// TwinCAT 3 PLC project PLC
// ProgramVersion: 3.1.4026.26
// libraries:
//   Tc2_Standard, * (Beckhoff Automation GmbH)
//   Tc2_System, * (Beckhoff Automation GmbH)
//   Tc2_Utilities, * (Beckhoff Automation GmbH)
//   Tc3_Database, * (Beckhoff Automation GmbH)
//   Tc3_EventLogger, * (Beckhoff Automation GmbH)
//   Tc3_JsonXml, * (Beckhoff Automation GmbH)
//   Tc3_IotBase, * (Beckhoff Automation GmbH)
//   TcUnit, * (www.tcunit.org)
// project tree:
//   / PlcTask.TcTTO, TestTask.TcTTO
//   POUs/ MAIN.TcPOU
//   POUs/fb/ FB_DfiRowBuffer.TcPOU, FB_DfiSampler.TcPOU, F_DfiNowString.TcPOU, FB_DfiCfgParse.TcPOU, FB_DfiConfigLoader.TcPOU, F_DfiSanitizeText.TcPOU, F_DfiStripSqlUnsafe.TcPOU, FB_DfiPayloadParser.TcPOU, FB_DfiSqlBuilder.TcPOU, FB_DfiDbWriter.TcPOU, FB_DfiMqttSubscriber.TcPOU
//   POUs/test/ PRG_DfiTests.TcPOU, FB_DfiRowBuffer_Tests.TcPOU, FB_DfiSampler_Tests.TcPOU, FB_DfiCfgParse_Tests.TcPOU, FB_DfiPayloadParser_Tests.TcPOU, FB_DfiSqlBuilder_Tests.TcPOU, F_DfiNowString_Tests.TcPOU, FB_DfiDbWriter_Fake.TcPOU, FB_DfiDbWriter_Tests.TcPOU
//   DUTs/ E_DfiRowKind.TcDUT, E_DfiWriterState.TcDUT, ST_EstoqueSnapshot.TcDUT, ST_EventoDfi.TcDUT, ST_DfiRow.TcDUT, ST_DfiConfig.TcDUT, ST_DfiDiag.TcDUT
//   GVLs/ GVL_Dfi.TcGVL
// real-time tasks:
//   TASK PlcTask: cycle T#100000us, priority 20, ADS port 350
//   TASK TestTask: cycle T#100000us, priority 21, ADS port 351

CONFIGURATION PLC
    RESOURCE PLC ON TwinCAT3
        TASK PlcTask(INTERVAL := T#10ms, PRIORITY := 1);
        TASK TestTask(INTERVAL := T#10ms, PRIORITY := 2);
        PROGRAM MAIN WITH PlcTask : MAIN;
        PROGRAM PRG_DfiTests WITH TestTask : PRG_DfiTests;
    END_RESOURCE
END_CONFIGURATION

// ---- DUTs/E_DfiRowKind.TcDUT
TYPE E_DfiRowKind :
(
	ESTOQUE_MUDANCA := 0,
	ESTOQUE_PERIODICO := 1,
	EVENTO := 2
) DINT;
END_TYPE

// ---- DUTs/E_DfiWriterState.TcDUT
TYPE E_DfiWriterState :
(
	IDLE := 0,
	CONNECT := 10,
	BUILD := 20,
	EXECUTE := 30,
	COMMIT := 40,
	ERROR := 90,
	DB_LOST := 99
) DINT;
END_TYPE

// ---- DUTs/ST_EstoqueSnapshot.TcDUT
TYPE ST_EstoqueSnapshot :
STRUCT
	nA : INT;
	nB : INT;
	nC : INT;
END_STRUCT
END_TYPE

// ---- DUTs/ST_EventoDfi.TcDUT
TYPE ST_EventoDfi :
STRUCT
	sEvento     : STRING(23);   // coluna eventos_hist.evento VARCHAR(24)
	sPeca       : STRING(1);    // 'A'|'B'|'C' ou '' (=> NULL)
	sDetalhe    : STRING(63);   // coluna detalhe VARCHAR(64)
	sPayloadRaw : STRING(254);  // coluna payload_raw VARCHAR(255)
END_STRUCT
END_TYPE

// ---- DUTs/ST_DfiRow.TcDUT
TYPE ST_DfiRow :
STRUCT
	eKind     : E_DfiRowKind;
	sTsPlc    : STRING(23);   // 'YYYY-MM-DD HH:MM:SS.mmm', carimbado no Push
	stEstoque : ST_EstoqueSnapshot;
	stEvento  : ST_EventoDfi;
END_STRUCT
END_TYPE

// ---- DUTs/ST_DfiConfig.TcDUT
TYPE ST_DfiConfig :
STRUCT
	sMqttHost     : STRING(120);
	nMqttPort     : UINT  := 1883;
	bUseTls       : BOOL  := FALSE;
	sCaCertPath   : STRING(255) := '/etc/ssl/certs/ca-certificates.crt';
	sMqttUser     : STRING(60);
	sMqttPass     : STRING(60);
	sTopicEstoque : STRING(120) := 'dataflow/estoque';
	sTopicEventos : STRING(120) := 'dataflow/eventos';
	nDbId         : UDINT := 1;
	tSamplePeriod : TIME  := T#60S;
	nBufferSize   : UDINT := 128;   // teto = FB_DfiRowBuffer.MAX_ROWS
	nEstoqueMax   : INT   := 999;
	bValid        : BOOL  := FALSE;   // TRUE após FB_DfiConfigLoader parsear o arquivo com sucesso
END_STRUCT
END_TYPE

// ---- DUTs/ST_DfiDiag.TcDUT
TYPE ST_DfiDiag :
STRUCT
	bConfigOk         : BOOL;
	bMqttConnected    : BOOL;
	bDbConnected      : BOOL;
	nReconnectCount   : UDINT;
	nBufferCount      : UDINT;
	nBufferHighWater  : UDINT;
	nBufferDropped    : ULINT;
	nRowsWritten      : ULINT;
	nDbErrors         : ULINT;
	nParseErrors      : ULINT;
	sUltimoParseError : STRING(120);
	sUltimoDbError    : STRING(255);
	eWriterState      : E_DfiWriterState;
END_STRUCT
END_TYPE

// ---- GVLs/GVL_Dfi.TcGVL
{attribute 'qualified_only'}
VAR_GLOBAL
	gCfg  : ST_DfiConfig;
	gDiag : ST_DfiDiag;
	// relogio de parede local (fonte do ts_plc; MAIN chama fbNow(bEnable := TRUE) todo ciclo)
	fbNow : Tc2_Utilities.FB_LocalSystemTime;
	// pipeline
	fbLoader  : FB_DfiConfigLoader;
	fbSub     : FB_DfiMqttSubscriber;
	fbParser  : FB_DfiPayloadParser;
	fbBuffer  : FB_DfiRowBuffer;
	fbSampler : FB_DfiSampler;
	fbWriter  : FB_DfiDbWriter;
END_VAR

// ---- POUs/MAIN.TcPOU
PROGRAM MAIN
VAR
	bBoot           : BOOL := TRUE;
	stUltimoEstoque : ST_EstoqueSnapshot;
	bEstoqueValido  : BOOL;
	bDiff           : BOOL;
	row             : ST_DfiRow;
END_VAR

// ---------------------------------------------------------------
// Orquestracao do historian DFI (Task 14). Pipeline por ciclo:
//   Config -> MQTT -> Parser -> Buffer -> Sampler -> DbWriter -> Diagnostico
// ---------------------------------------------------------------

// Relogio de parede local: ticado todo ciclo (independe da config) para que
// F_DfiNowString() tenha um TIMESTRUCT valido. Leva alguns ciclos ate bValid.
GVL_Dfi.fbNow(bEnable := TRUE);

// 0. Config (uma vez no arranque; retenta se falhar)
IF bBoot THEN
	GVL_Dfi.fbLoader(bExecute := TRUE, sPath := '/etc/dfi/historian.conf');
	IF GVL_Dfi.fbLoader.bDone THEN
		bBoot := FALSE;
		IF NOT GVL_Dfi.fbLoader.bError AND GVL_Dfi.fbLoader.stCfg.bValid THEN
			GVL_Dfi.gCfg := GVL_Dfi.fbLoader.stCfg;
		END_IF
	END_IF
END_IF
GVL_Dfi.gDiag.bConfigOk := GVL_Dfi.gCfg.bValid;
IF NOT GVL_Dfi.gCfg.bValid THEN
	RETURN;   // sem config valida, nao conecta em nada
END_IF

GVL_Dfi.fbBuffer(nCapacity := GVL_Dfi.gCfg.nBufferSize);

// 1. MQTT
GVL_Dfi.fbSub(stConfig := GVL_Dfi.gCfg, bEnable := TRUE);

// 2. Parse + roteamento
IF GVL_Dfi.fbSub.bNewMessage THEN
	GVL_Dfi.fbParser(bExecute := TRUE,
	                 sTopic   := GVL_Dfi.fbSub.sTopic,
	                 sPayload := GVL_Dfi.fbSub.sPayload,
	                 stConfig := GVL_Dfi.gCfg);
	IF GVL_Dfi.fbParser.bOk THEN
		// Limpa a linha reutilizada antes de montar (row e VAR persistente do MAIN).
		row.sTsPlc              := '';
		row.stEstoque.nA        := 0;
		row.stEstoque.nB        := 0;
		row.stEstoque.nC        := 0;
		row.stEvento.sEvento    := '';
		row.stEvento.sPeca      := '';
		row.stEvento.sDetalhe   := '';
		row.stEvento.sPayloadRaw := '';
		CASE GVL_Dfi.fbParser.eKind OF
			E_DfiRowKind.ESTOQUE_MUDANCA:
				stUltimoEstoque := GVL_Dfi.fbParser.stEstoque;
				bEstoqueValido  := TRUE;
				bDiff := (NOT GVL_Dfi.fbWriter.bUltimoGravadoValido)
				      OR (GVL_Dfi.fbParser.stEstoque.nA <> GVL_Dfi.fbWriter.stUltimoGravado.nA)
				      OR (GVL_Dfi.fbParser.stEstoque.nB <> GVL_Dfi.fbWriter.stUltimoGravado.nB)
				      OR (GVL_Dfi.fbParser.stEstoque.nC <> GVL_Dfi.fbWriter.stUltimoGravado.nC);
				IF bDiff THEN
					row.eKind     := E_DfiRowKind.ESTOQUE_MUDANCA;
					row.sTsPlc    := F_DfiNowString();
					row.stEstoque := GVL_Dfi.fbParser.stEstoque;
					GVL_Dfi.fbBuffer.Push(row);
				END_IF

			E_DfiRowKind.EVENTO:
				row.eKind    := E_DfiRowKind.EVENTO;
				row.sTsPlc   := F_DfiNowString();
				row.stEvento := GVL_Dfi.fbParser.stEvento;
				GVL_Dfi.fbBuffer.Push(row);
		END_CASE
	ELSE
		GVL_Dfi.gDiag.nParseErrors      := GVL_Dfi.gDiag.nParseErrors + 1;
		GVL_Dfi.gDiag.sUltimoParseError := GVL_Dfi.fbParser.sParseError;
	END_IF
	GVL_Dfi.fbParser(bExecute := FALSE);   // rearma a borda de subida
END_IF

// 3. Amostra periodica
GVL_Dfi.fbSampler(stUltimoEstoque := stUltimoEstoque,
                  bValido         := bEstoqueValido,
                  tPeriodo        := GVL_Dfi.gCfg.tSamplePeriod,
                  fbBuffer        := GVL_Dfi.fbBuffer);

// 4. Dreno para o banco
GVL_Dfi.fbWriter(stConfig := GVL_Dfi.gCfg, fbBuffer := GVL_Dfi.fbBuffer);

// 5. Diagnostico
GVL_Dfi.gDiag.bMqttConnected   := GVL_Dfi.fbSub.bConnected;
GVL_Dfi.gDiag.nReconnectCount  := GVL_Dfi.fbSub.nReconnectCount;
GVL_Dfi.gDiag.bDbConnected     := GVL_Dfi.fbWriter.bDbConnected;
GVL_Dfi.gDiag.eWriterState     := GVL_Dfi.fbWriter.eState;
GVL_Dfi.gDiag.nRowsWritten     := GVL_Dfi.fbWriter.nRowsWritten;
GVL_Dfi.gDiag.nDbErrors        := GVL_Dfi.fbWriter.nErrors;
GVL_Dfi.gDiag.sUltimoDbError   := GVL_Dfi.fbWriter.sLastError;
GVL_Dfi.gDiag.nBufferCount     := GVL_Dfi.fbBuffer.nCount;
GVL_Dfi.gDiag.nBufferHighWater := GVL_Dfi.fbBuffer.nHighWater;
GVL_Dfi.gDiag.nBufferDropped   := GVL_Dfi.fbBuffer.nDropped;

END_PROGRAM

// ---- POUs/fb/F_DfiNowString.TcPOU
FUNCTION F_DfiNowString : STRING(23)
VAR_INPUT
END_VAR
VAR
	fbGetSystemTime : Tc2_Utilities.GETSYSTEMTIME;
	ft              : T_FILETIME;
	tmst            : TIMESTRUCT;
	nYear : INT;
	nMon  : INT;
	nDay  : INT;
	nHour : INT;
	nMin  : INT;
	nSec  : INT;
	nMs   : INT;
	sYear : STRING(4);
	sMon  : STRING(2);
	sDay  : STRING(2);
	sHour : STRING(2);
	sMin  : STRING(2);
	sSec  : STRING(2);
	sMs   : STRING(3);
END_VAR

// Retorna o instante atual como 'YYYY-MM-DD HH:MM:SS.mmm' (23 chars). Fonte: Tc2_Utilities.GETSYSTEMTIME + FILETIME_TO_SYSTEMTIME (UTC).
// TODO: local timezone conversion (RT Linux timedatectl sets TZ; verify UTC vs local at bench)
fbGetSystemTime(timeLoDW => ft.dwLowDateTime, timeHiDW => ft.dwHighDateTime);
FILETIME_TO_SYSTEMTIME(fileTime := ft);

nYear := TO_INT(tmst.wYear);
nMon  := TO_INT(tmst.wMonth);
nDay  := TO_INT(tmst.wDay);
nHour := TO_INT(tmst.wHour);
nMin  := TO_INT(tmst.wMinute);
nSec  := TO_INT(tmst.wSecond);
nMs   := TO_INT(tmst.wMilliseconds);

sYear := INT_TO_STRING(nYear);

IF nMon < 10 THEN sMon := CONCAT('0', INT_TO_STRING(nMon)); ELSE sMon := INT_TO_STRING(nMon); END_IF
IF nDay < 10 THEN sDay := CONCAT('0', INT_TO_STRING(nDay)); ELSE sDay := INT_TO_STRING(nDay); END_IF
IF nHour < 10 THEN sHour := CONCAT('0', INT_TO_STRING(nHour)); ELSE sHour := INT_TO_STRING(nHour); END_IF
IF nMin < 10 THEN sMin := CONCAT('0', INT_TO_STRING(nMin)); ELSE sMin := INT_TO_STRING(nMin); END_IF
IF nSec < 10 THEN sSec := CONCAT('0', INT_TO_STRING(nSec)); ELSE sSec := INT_TO_STRING(nSec); END_IF

IF nMs < 10 THEN
	sMs := CONCAT('00', INT_TO_STRING(nMs));
ELSIF nMs < 100 THEN
	sMs := CONCAT('0', INT_TO_STRING(nMs));
ELSE
	sMs := INT_TO_STRING(nMs);
END_IF

F_DfiNowString := CONCAT(sYear, '-');
F_DfiNowString := CONCAT(F_DfiNowString, sMon);
F_DfiNowString := CONCAT(F_DfiNowString, '-');
F_DfiNowString := CONCAT(F_DfiNowString, sDay);
F_DfiNowString := CONCAT(F_DfiNowString, ' ');
F_DfiNowString := CONCAT(F_DfiNowString, sHour);
F_DfiNowString := CONCAT(F_DfiNowString, ':');
F_DfiNowString := CONCAT(F_DfiNowString, sMin);
F_DfiNowString := CONCAT(F_DfiNowString, ':');
F_DfiNowString := CONCAT(F_DfiNowString, sSec);
F_DfiNowString := CONCAT(F_DfiNowString, '.');
F_DfiNowString := CONCAT(F_DfiNowString, sMs);

END_FUNCTION

// ---- POUs/test/PRG_DfiTests.TcPOU
PROGRAM PRG_DfiTests
VAR
	fbRowBufferTests : FB_DfiRowBuffer_Tests;
	// suites added by later tasks:
	fbSamplerTests   : FB_DfiSampler_Tests;
	fbCfgParseTests  : FB_DfiCfgParse_Tests;
	fbParserTests    : FB_DfiPayloadParser_Tests;
	fbSqlBuilderTests: FB_DfiSqlBuilder_Tests;
	fbNowStringTests : F_DfiNowString_Tests;
	fbDbWriterTests  : FB_DfiDbWriter_Tests;
END_VAR

TcUnit.RUN();

END_PROGRAM

// ---- POUs/test/FB_DfiRowBuffer_Tests.TcPOU
FUNCTION_BLOCK FB_DfiRowBuffer_Tests EXTENDS TcUnit.FB_TestSuite
VAR
END_VAR

Test_PushPop_PreservaOrdemFIFO();
Test_Peek_NaoRemove();
Test_PopVazio_RetornaFalse();
Test_Overflow_DescartaMaisAntigo_IncrementaDropped();
Test_HighWater_AcompanhaPico();

METHOD PRIVATE Test_HighWater_AcompanhaPico
VAR
	fb : FB_DfiRowBuffer := (nCapacity := 8);
	linha : ST_DfiRow;
	i : INT;
END_VAR
TEST('HighWater_AcompanhaPico');
FOR i := 1 TO 5 DO fb.Push(linha); END_FOR
fb.Pop(); fb.Pop();
AssertEquals_UDINT(Expected := 3, Actual := fb.nCount, Message := 'nCount 3 apos 2 Pop');
AssertEquals_UDINT(Expected := 5, Actual := fb.nHighWater, Message := 'highwater guarda o pico 5');
TEST_FINISHED();
END_METHOD

METHOD PRIVATE Test_Overflow_DescartaMaisAntigo_IncrementaDropped
VAR
	fb : FB_DfiRowBuffer := (nCapacity := 3);
	linha, out : ST_DfiRow;
	i : INT;
	okPush : BOOL;
END_VAR
TEST('Overflow_DescartaMaisAntigo_IncrementaDropped');
FOR i := 1 TO 3 DO
	linha.stEstoque.nA := i; fb.Push(linha);
END_FOR
linha.stEstoque.nA := 4;
okPush := fb.Push(linha);                       // capacidade estourada
AssertFalse(okPush, 'Push retorna FALSE ao descartar');
AssertEquals_ULINT(Expected := 1, Actual := fb.nDropped, Message := 'nDropped incrementa');
AssertEquals_UDINT(Expected := 3, Actual := fb.nCount, Message := 'nCount fica no teto');
fb.Peek();
AssertEquals_INT(Expected := 2, Actual := out.stEstoque.nA, Message := 'frente agora eh o 2o (1o descartado)');
TEST_FINISHED();
END_METHOD

METHOD PRIVATE Test_Peek_NaoRemove
VAR
	fb : FB_DfiRowBuffer := (nCapacity := 4);
	a, out : ST_DfiRow;
	ok : BOOL;
END_VAR
TEST('Peek_NaoRemove');
a.eKind := E_DfiRowKind.ESTOQUE_MUDANCA; a.stEstoque.nA := 7;
fb.Push(a);
ok := fb.Peek();
AssertTrue(ok, 'Peek TRUE com 1 item');
AssertEquals_INT(Expected := 7, Actual := out.stEstoque.nA, Message := 'valor via Peek');
AssertEquals_UDINT(Expected := 1, Actual := fb.nCount, Message := 'Peek nao remove');
TEST_FINISHED();
END_METHOD

METHOD PRIVATE Test_PopVazio_RetornaFalse
VAR
	fb : FB_DfiRowBuffer := (nCapacity := 4);
	out : ST_DfiRow;
END_VAR
TEST('PopVazio_RetornaFalse');
AssertFalse(fb.Peek(), 'Peek FALSE vazio');
AssertFalse(fb.Pop(), 'Pop FALSE vazio');
TEST_FINISHED();
END_METHOD

METHOD PRIVATE Test_PushPop_PreservaOrdemFIFO
VAR
	fb : FB_DfiRowBuffer := (nCapacity := 4);
	a, b, out : ST_DfiRow;
END_VAR
TEST('PushPop_PreservaOrdemFIFO');
a.eKind := E_DfiRowKind.EVENTO; a.stEvento.sEvento := 'entrega';
b.eKind := E_DfiRowKind.EVENTO; b.stEvento.sEvento := 'erro';
fb.Push(a); fb.Push(b);
AssertEquals_UDINT(Expected := 2, Actual := fb.nCount, Message := 'nCount apos 2 Push');
fb.Peek(); fb.Pop();
AssertEquals_STRING(Expected := 'entrega', Actual := out.stEvento.sEvento, Message := '1o a sair');
fb.Peek(); fb.Pop();
AssertEquals_STRING(Expected := 'erro', Actual := out.stEvento.sEvento, Message := '2o a sair');
AssertEquals_UDINT(Expected := 0, Actual := fb.nCount, Message := 'vazio ao final');
TEST_FINISHED();
END_METHOD

END_FUNCTION_BLOCK

// ---- POUs/fb/FB_DfiRowBuffer.TcPOU
FUNCTION_BLOCK FB_DfiRowBuffer
VAR_INPUT
	nCapacity : UDINT := 128;
END_VAR
VAR_OUTPUT
	nCount     : UDINT;
	nHighWater : UDINT;
	nDropped   : ULINT;
END_VAR
VAR CONSTANT
	// Teto fisico do array. ST_DfiRow ~380 bytes -> 128 linhas ~= 49 KB.
	// Nao aumentar sem necessidade: as suites TcUnit declaram FB_DfiRowBuffer
	// como local de metodo (vai para a pilha da task) e 512 linhas (~195 KB)
	// estouram a pilha da TestTask. 128 linhas = ~2 min de store-and-forward.
	MAX_ROWS : UDINT := 128;   // nCapacity <= MAX_ROWS
END_VAR
VAR
	aRows  : ARRAY[0..MAX_ROWS-1] OF ST_DfiRow;
	nHead  : UDINT;            // índice de leitura (frente)
	nTail  : UDINT;            // índice de escrita (próxima posição livre)
	nCap   : UDINT;            // capacidade efetiva (clamp de nCapacity)
	bInit  : BOOL;
END_VAR

IF NOT bInit THEN
	nCap := LIMIT(1, nCapacity, MAX_ROWS);
	bInit := TRUE;
END_IF
// nCount é mantido pelos métodos; corpo do FB é no-op.

METHOD Push : BOOL
VAR_INPUT
	stRow : ST_DfiRow;
END_VAR
VAR
	bClean : BOOL;
END_VAR
IF NOT bInit THEN nCap := LIMIT(1, nCapacity, MAX_ROWS); bInit := TRUE; END_IF
bClean := TRUE;
IF nCount >= nCap THEN
	// buffer cheio: descarta o mais antigo
	nHead := (nHead + 1) MOD nCap;
	nCount := nCount - 1;
	nDropped := nDropped + 1;
	bClean := FALSE;
END_IF
aRows[nTail] := stRow;
nTail := (nTail + 1) MOD nCap;
nCount := nCount + 1;
IF nCount > nHighWater THEN nHighWater := nCount; END_IF
Push := bClean;
END_METHOD

METHOD Peek : BOOL
VAR_OUTPUT
	stRow : ST_DfiRow;
END_VAR
IF nCount = 0 THEN
	Peek := FALSE;
	RETURN;
END_IF
stRow := aRows[nHead];
Peek := TRUE;
END_METHOD

METHOD Pop : BOOL
IF nCount = 0 THEN
	Pop := FALSE;
	RETURN;
END_IF
nHead := (nHead + 1) MOD nCap;
nCount := nCount - 1;
Pop := TRUE;
END_METHOD

END_FUNCTION_BLOCK

// ---- POUs/test/FB_DfiSampler_Tests.TcPOU
FUNCTION_BLOCK FB_DfiSampler_Tests EXTENDS TcUnit.FB_TestSuite
VAR
END_VAR

Test_NaoDispara_SemEstoqueValido();
Test_Dispara_AposPeriodo_ComUltimoEstoque();
Test_Rearma_ACadaPeriodo();

METHOD PRIVATE Test_Dispara_AposPeriodo_ComUltimoEstoque
VAR
	fbBuf : FB_DfiRowBuffer := (nCapacity := 8);
	fbSut : FB_DfiSampler;
	est   : ST_EstoqueSnapshot;
	out   : ST_DfiRow;
END_VAR
TEST('Dispara_AposPeriodo_ComUltimoEstoque');
est.nA := 3; est.nB := 4; est.nC := 5;
// simula passagem de tempo: TcUnit roda em ciclos; usa CycleCallCount + tPeriodo curto
fbSut(stUltimoEstoque := est, bValido := TRUE, tPeriodo := T#20MS, fbBuffer := fbBuf);
// esperar o TON: chamar o SUT em ciclos sucessivos até nCount = 1 ou timeout do teste
// (TcUnit avança o tempo real entre ciclos da task de teste)
IF fbBuf.nCount >= 1 THEN
	fbBuf.Peek();
	AssertEquals_INT(Expected := 3, Actual := out.stEstoque.nA, Message := 'snapshot A');
	AssertTrue(out.eKind = E_DfiRowKind.ESTOQUE_PERIODICO, 'eKind periodico');
	TEST_FINISHED();
END_IF
END_METHOD

METHOD PRIVATE Test_NaoDispara_SemEstoqueValido
VAR
	fbBuf : FB_DfiRowBuffer := (nCapacity := 8);
	fbSut : FB_DfiSampler;
	est   : ST_EstoqueSnapshot;
	i     : INT;
END_VAR
TEST('NaoDispara_SemEstoqueValido');
FOR i := 1 TO 50 DO
	fbSut(stUltimoEstoque := est, bValido := FALSE, tPeriodo := T#100MS, fbBuffer := fbBuf);
END_FOR
AssertEquals_UDINT(Expected := 0, Actual := fbBuf.nCount, Message := 'nada empurrado sem estoque valido');
TEST_FINISHED();
END_METHOD

METHOD PRIVATE Test_Rearma_ACadaPeriodo
VAR
	fbBuf : FB_DfiRowBuffer := (nCapacity := 8);
	fbSut : FB_DfiSampler;
	est   : ST_EstoqueSnapshot;
END_VAR
TEST('Rearma_ACadaPeriodo');
est.nA := 1; est.nB := 2; est.nC := 3;
// TcUnit re-roda este metodo a cada ciclo ate TEST_FINISHED(); o TON avanca com o tempo real.
// Apos o 1o push o SUT rearma sozinho e continua empurrando a cada tPeriodo.
fbSut(stUltimoEstoque := est, bValido := TRUE, tPeriodo := T#20MS, fbBuffer := fbBuf);
IF fbBuf.nCount >= 2 THEN
	AssertTrue(fbBuf.nCount >= 2, 'rearmou e empurrou pelo menos 2x');
	AssertTrue(fbSut.nPushed = fbBuf.nCount, 'nPushed acompanha nCount (sem descartes)');
	TEST_FINISHED();
END_IF
END_METHOD

END_FUNCTION_BLOCK

// ---- POUs/fb/FB_DfiSampler.TcPOU
FUNCTION_BLOCK FB_DfiSampler
VAR_INPUT
	stUltimoEstoque : ST_EstoqueSnapshot;
	bValido         : BOOL;
	tPeriodo        : TIME;
END_VAR
VAR_IN_OUT
	fbBuffer : FB_DfiRowBuffer;
END_VAR
VAR_OUTPUT
	nPushed : ULINT;
END_VAR
VAR
	fbTon : TON;
	row   : ST_DfiRow;
END_VAR

fbTon(IN := bValido, PT := tPeriodo);
IF fbTon.Q THEN
	fbTon(IN := FALSE);           // rearma
	row.eKind := E_DfiRowKind.ESTOQUE_PERIODICO;
	row.stEstoque := stUltimoEstoque;
	row.sTsPlc := F_DfiNowString();   // helper da Task 10, ver nota
	fbBuffer.Push(row);
	nPushed := nPushed + 1;
END_IF

END_FUNCTION_BLOCK

// ---- POUs/test/FB_DfiCfgParse_Tests.TcPOU
FUNCTION_BLOCK FB_DfiCfgParse_Tests EXTENDS TcUnit.FB_TestSuite
VAR
END_VAR

Test_ParseLine_MapeiaChavesConhecidas();
Test_ParseLine_ComentarioEBranco_NoOp();
Test_ParseLine_ChaveDesconhecida_RetornaFalse();
Test_ParseText_ExemploCompleto_ValidaEbValidTrue();
Test_ParseText_SemHost_bValidFalse();

METHOD PRIVATE Test_ParseLine_ChaveDesconhecida_RetornaFalse
VAR
	fb  : FB_DfiCfgParse;
	cfg : ST_DfiConfig;
END_VAR
TEST('ParseLine_ChaveDesconhecida_RetornaFalse');
AssertFalse(fb.ParseLine('foo=bar', cfg), 'chave desconhecida => FALSE');
AssertFalse(fb.ParseLine('mqtt_port=abc', cfg), 'valor nao-numerico => FALSE');
TEST_FINISHED();
END_METHOD

METHOD PRIVATE Test_ParseLine_ComentarioEBranco_NoOp
VAR
	fb  : FB_DfiCfgParse;
	cfg : ST_DfiConfig;
END_VAR
TEST('ParseLine_ComentarioEBranco_NoOp');
AssertTrue(fb.ParseLine('# comentario', cfg), 'comentario ok');
AssertTrue(fb.ParseLine('', cfg), 'linha vazia ok');
AssertTrue(fb.ParseLine('   ', cfg), 'espacos ok');
AssertEquals_STRING(Expected := '', Actual := cfg.sMqttHost, Message := 'nada mudou');
TEST_FINISHED();
END_METHOD

METHOD PRIVATE Test_ParseLine_MapeiaChavesConhecidas
VAR
	fb  : FB_DfiCfgParse;
	cfg : ST_DfiConfig;
END_VAR
TEST('ParseLine_MapeiaChavesConhecidas');
fb.ParseLine('mqtt_host=10.0.0.5', cfg);
fb.ParseLine('mqtt_port=8883', cfg);
fb.ParseLine('mqtt_use_tls=1', cfg);
fb.ParseLine('sample_period_s=30', cfg);
fb.ParseLine('buffer_size=256', cfg);
fb.ParseLine('estoque_max=50', cfg);
AssertEquals_STRING(Expected := '10.0.0.5', Actual := cfg.sMqttHost, Message := 'host');
AssertEquals_UINT(Expected := 8883, Actual := cfg.nMqttPort, Message := 'port');
AssertTrue(cfg.bUseTls, 'tls');
AssertTrue(cfg.tSamplePeriod = T#30S, 'periodo');
AssertEquals_UDINT(Expected := 256, Actual := cfg.nBufferSize, Message := 'buffer');
AssertEquals_INT(Expected := 50, Actual := cfg.nEstoqueMax, Message := 'estoque_max');
TEST_FINISHED();
END_METHOD

METHOD PRIVATE Test_ParseText_ExemploCompleto_ValidaEbValidTrue
VAR
	fb  : FB_DfiCfgParse;
	cfg : ST_DfiConfig;
	conjunto   : STRING(4095);
END_VAR
TEST('ParseText_ExemploCompleto');
conjunto := CONCAT('mqtt_host=192.168.0.50$N', CONCAT('mqtt_port=1883$N', CONCAT('topic_estoque=dataflow/estoque$N', 'db_id=1$N')));
AssertTrue(fb.ParseText(conjunto, cfg), 'ParseText ok');
AssertTrue(cfg.bValid, 'bValid TRUE com host preenchido');
AssertEquals_STRING(Expected := 'dataflow/estoque', Actual := cfg.sTopicEstoque, Message := 'topico');
TEST_FINISHED();
END_METHOD

METHOD PRIVATE Test_ParseText_SemHost_bValidFalse
VAR
	fb  : FB_DfiCfgParse;
	cfg : ST_DfiConfig;
END_VAR
TEST('ParseText_SemHost_bValidFalse');
fb.ParseText('mqtt_port=1883$Ndb_id=1', cfg);
AssertFalse(cfg.bValid, 'sem host => invalido');
TEST_FINISHED();
END_METHOD

END_FUNCTION_BLOCK

// ---- POUs/fb/FB_DfiCfgParse.TcPOU
FUNCTION_BLOCK FB_DfiCfgParse
VAR
END_VAR

// Sem lógica no corpo do FB: o parsing é feito pelos métodos ParseLine / ParseText.

METHOD PRIVATE AllDigits : BOOL
VAR_INPUT
	sEntrada : STRING(255);
END_VAR
VAR
	i    : INT;
	nLen : INT;
	c    : BYTE;
	p    : POINTER TO BYTE;
	Sinal: STRING;
END_VAR
// TRUE somente se sIn não estiver vazia e for composta apenas por '0'..'9'.
nLen := LEN(sEntrada);
IF nLen = 0 THEN
	AllDigits := FALSE;
	RETURN;
END_IF
p := ADR(sEntrada);
FOR i := 0 TO nLen - 1 DO
	c := p[i];
	IF (c < 16#30) OR (c > 16#39) THEN
		AllDigits := FALSE;
		RETURN;
	END_IF
END_FOR
AllDigits := TRUE;
END_METHOD

METHOD ParseLine : BOOL
VAR_INPUT
	sLine : STRING(255);
END_VAR
VAR_IN_OUT
	stCfg : ST_DfiConfig;
END_VAR
VAR
	sWork : STRING(255);
	sKey  : STRING(255);
	sVal  : STRING(255);
	nEq   : INT;
	nLen  : INT;
	nBuf  : UDINT;
END_VAR
// --- normaliza: trim de espaços/tabs nas duas pontas ---
sWork := THIS^.TrimBoth(sLine);
nLen  := LEN(sWork);

// --- linha vazia ou comentário => no-op com sucesso ---
IF nLen = 0 THEN
	ParseLine := TRUE;
	RETURN;
END_IF
IF LEFT(sWork, 1) = '#' THEN
	ParseLine := TRUE;
	RETURN;
END_IF

// --- precisa ter '=' ---
nEq := FIND(sWork, '=');
IF nEq = 0 THEN
	ParseLine := FALSE;
	RETURN;
END_IF

// --- separa chave / valor e faz trim dos dois ---
sKey := THIS^.TrimBoth(LEFT(sWork, nEq - 1));
sVal := THIS^.TrimBoth(RIGHT(sWork, nLen - nEq));

// --- CASE de string não é permitido em ST: cadeia de IF/ELSIF ---
IF sKey = 'mqtt_host' THEN
	stCfg.sMqttHost := sVal;

ELSIF sKey = 'mqtt_port' THEN
	IF NOT THIS^.AllDigits(sVal) THEN
		ParseLine := FALSE;
		RETURN;
	END_IF
	stCfg.nMqttPort := STRING_TO_UINT(sVal);

ELSIF sKey = 'mqtt_use_tls' THEN
	// aceita qualquer valor: '1' => TRUE, qualquer outra coisa => FALSE
	stCfg.bUseTls := (sVal = '1');

ELSIF sKey = 'mqtt_ca_cert_path' THEN
	stCfg.sCaCertPath := sVal;

ELSIF sKey = 'mqtt_user' THEN
	stCfg.sMqttUser := sVal;

ELSIF sKey = 'mqtt_pass' THEN
	stCfg.sMqttPass := sVal;

ELSIF sKey = 'topic_estoque' THEN
	stCfg.sTopicEstoque := sVal;

ELSIF sKey = 'topic_eventos' THEN
	stCfg.sTopicEventos := sVal;

ELSIF sKey = 'db_id' THEN
	IF NOT THIS^.AllDigits(sVal) THEN
		ParseLine := FALSE;
		RETURN;
	END_IF
	stCfg.nDbId := STRING_TO_UDINT(sVal);

ELSIF sKey = 'sample_period_s' THEN
	IF NOT THIS^.AllDigits(sVal) THEN
		ParseLine := FALSE;
		RETURN;
	END_IF
	stCfg.tSamplePeriod := UDINT_TO_TIME(STRING_TO_UDINT(sVal) * 1000);

ELSIF sKey = 'buffer_size' THEN
	IF NOT THIS^.AllDigits(sVal) THEN
		ParseLine := FALSE;
		RETURN;
	END_IF
	nBuf := STRING_TO_UDINT(sVal);
	IF nBuf < 1 THEN
		nBuf := 1;
	END_IF
	IF nBuf > 512 THEN
		nBuf := 512;
	END_IF
	stCfg.nBufferSize := nBuf;

ELSIF sKey = 'estoque_max' THEN
	IF NOT THIS^.AllDigits(sVal) THEN
		ParseLine := FALSE;
		RETURN;
	END_IF
	stCfg.nEstoqueMax := STRING_TO_INT(sVal);

ELSE
	// chave desconhecida
	ParseLine := FALSE;
	RETURN;
END_IF

ParseLine := TRUE;
END_METHOD

METHOD ParseText : BOOL
VAR_INPUT
	sText : STRING(4095);
END_VAR
VAR_IN_OUT
	stCfg : ST_DfiConfig;
END_VAR
VAR
	bAllOk : BOOL;
	i      : INT;
	j      : INT;
	nEnd   : INT;
	nStart : INT;
	nCnt   : INT;
	p      : POINTER TO BYTE;
	pFrag  : POINTER TO BYTE;
	sFrag  : STRING(255);
END_VAR
// Quebra sText em linhas por $N (LF, 16#0A) e $R (CR, 16#0D).
// Trata $R$N, $N sozinho e $R sozinho; fragmentos vazios são ignorados.
// Varredura por ponteiro de bytes (as funções string padrão do Tc2_Standard
// operam em STRING(255) e truncariam sText, que é STRING(4095)).
bAllOk := TRUE;
p      := ADR(sText);
pFrag  := ADR(sFrag);

// comprimento real: varre até o NUL, com teto no tamanho do buffer
nEnd := 0;
WHILE (nEnd < 4095) AND (p[nEnd] <> 0) DO
	nEnd := nEnd + 1;
END_WHILE

nStart := 0;
FOR i := 0 TO nEnd DO
	// i = nEnd força o flush do último fragmento (arquivo sem quebra no fim)
	IF (i = nEnd) OR (p[i] = 16#0A) OR (p[i] = 16#0D) THEN
		nCnt := i - nStart;
		IF nCnt > 0 THEN
			IF nCnt > 254 THEN
				nCnt := 254;
			END_IF
			FOR j := 0 TO nCnt - 1 DO
				pFrag[j] := p[nStart + j];
			END_FOR
			pFrag[nCnt] := 0;
			IF NOT ParseLine(sFrag, stCfg) THEN
				bAllOk := FALSE;
			END_IF
		END_IF
		nStart := i + 1;
	END_IF
END_FOR

stCfg.bValid := bAllOk AND (stCfg.sMqttHost <> '');
ParseText := bAllOk;
END_METHOD

METHOD PRIVATE TrimBoth : STRING(255)
VAR_INPUT
	sEntrada : STRING(255);
END_VAR
VAR
	nLen   : INT;
	nStart : INT;
	nEnd   : INT;
	c      : BYTE;
	p      : POINTER TO BYTE;
END_VAR
// Remove espaços (16#20) e tabs (16#09) do início e do fim.
nLen := LEN(sEntrada);
IF nLen = 0 THEN
	TrimBoth := '';
	RETURN;
END_IF
p := ADR(sEntrada);

nStart := 0;
WHILE (nStart < nLen) AND ((p[nStart] = 16#20) OR (p[nStart] = 16#09)) DO
	nStart := nStart + 1;
END_WHILE
IF nStart >= nLen THEN
	TrimBoth := '';
	RETURN;
END_IF

nEnd := nLen - 1;
WHILE (nEnd > nStart) AND ((p[nEnd] = 16#20) OR (p[nEnd] = 16#09)) DO
	nEnd := nEnd - 1;
END_WHILE

TrimBoth := MID(sEntrada, nEnd - nStart + 1, nStart + 1);
END_METHOD

END_FUNCTION_BLOCK

// ---- POUs/test/FB_DfiPayloadParser_Tests.TcPOU
FUNCTION_BLOCK FB_DfiPayloadParser_Tests EXTENDS TcUnit.FB_TestSuite
VAR
END_VAR

Test_Estoque_Valido();
Test_Evento_Entrega();
Test_Evento_ErroTimeout_MapeiaTipoParaDetalhe();
Test_JsonInvalido_bOkFalse();
Test_TypeAusente_bOkFalse();
Test_TypeDesconhecido_bOkFalse();
Test_Estoque_CampoFaltando_bOkFalse();
Test_Estoque_Negativo_bOkFalse();
Test_Estoque_AcimaDoMax_bOkFalse();
Test_Evento_SemCampoEvento_bOkFalse();
Test_Evento_PecaInvalida_bOkFalse();
Test_Evento_PecaAusente_Ok_PecaVazia();
Test_Evento_DetalheComAspa_bOkFalse();
Test_Evento_EventoComPontoEVirgula_bOkFalse();
Test_Evento_DetalheLongo_Truncado();
Test_Evento_PayloadRaw_Preenchido();
Test_TopicoDesconhecido_bOkFalse();
Test_StripSqlUnsafe_RemoveAspas();

METHOD PRIVATE Test_Estoque_Valido
VAR
	fb  : FB_DfiPayloadParser;
	cfg : ST_DfiConfig;
END_VAR
TEST('Estoque_Valido');
cfg.sTopicEstoque := 'dataflow/estoque'; cfg.nEstoqueMax := 999;
fb(bExecute := TRUE, sTopic := 'dataflow/estoque',
   sPayload := '{"type":"estoque","pecaA":4,"pecaB":5,"pecaC":6}', stConfig := cfg);
AssertTrue(fb.bOk, 'bOk');
AssertTrue(fb.eKind = E_DfiRowKind.ESTOQUE_MUDANCA, 'eKind');
AssertEquals_INT(4, fb.stEstoque.nA, 'A'); AssertEquals_INT(5, fb.stEstoque.nB, 'B'); AssertEquals_INT(6, fb.stEstoque.nC, 'C');
TEST_FINISHED();
END_METHOD

METHOD PRIVATE Test_Evento_Entrega
VAR
	fb  : FB_DfiPayloadParser;
	cfg : ST_DfiConfig;
END_VAR
TEST('Evento_Entrega');
cfg.sTopicEventos := 'dataflow/eventos';
fb(bExecute := TRUE, sTopic := 'dataflow/eventos',
   sPayload := '{"type":"evento","evento":"entrega","peca":"A"}', stConfig := cfg);
AssertTrue(fb.bOk, 'bOk');
AssertTrue(fb.eKind = E_DfiRowKind.EVENTO, 'eKind');
AssertEquals_STRING('entrega', fb.stEvento.sEvento, 'evento');
AssertEquals_STRING('A', fb.stEvento.sPeca, 'peca');
AssertEquals_STRING('', fb.stEvento.sDetalhe, 'sem detalhe');
TEST_FINISHED();
END_METHOD

METHOD PRIVATE Test_Evento_ErroTimeout_MapeiaTipoParaDetalhe
VAR
	fb  : FB_DfiPayloadParser;
	cfg : ST_DfiConfig;
END_VAR
TEST('Evento_ErroTimeout');
cfg.sTopicEventos := 'dataflow/eventos';
fb(bExecute := TRUE, sTopic := 'dataflow/eventos',
   sPayload := '{"type":"evento","evento":"erro","tipo":"timeout","peca":"B"}', stConfig := cfg);
AssertTrue(fb.bOk, 'bOk');
AssertEquals_STRING('erro', fb.stEvento.sEvento, 'evento');
AssertEquals_STRING('timeout', fb.stEvento.sDetalhe, 'tipo -> detalhe');
AssertEquals_STRING('B', fb.stEvento.sPeca, 'peca');
TEST_FINISHED();
END_METHOD

METHOD PRIVATE Test_JsonInvalido_bOkFalse
VAR
	fb  : FB_DfiPayloadParser;
	cfg : ST_DfiConfig;
END_VAR
TEST('JsonInvalido_bOkFalse');
cfg.sTopicEstoque := 'dataflow/estoque';
fb(bExecute := TRUE, sTopic := 'dataflow/estoque',
   sPayload := '{not json', stConfig := cfg);
AssertFalse(fb.bOk, 'bOk FALSE');
AssertEquals_STRING('json', fb.sParseError, 'sParseError');
TEST_FINISHED();
END_METHOD

METHOD PRIVATE Test_TypeAusente_bOkFalse
VAR
	fb  : FB_DfiPayloadParser;
	cfg : ST_DfiConfig;
END_VAR
TEST('TypeAusente_bOkFalse');
cfg.sTopicEstoque := 'dataflow/estoque';
fb(bExecute := TRUE, sTopic := 'dataflow/estoque',
   sPayload := '{"pecaA":1}', stConfig := cfg);
AssertFalse(fb.bOk, 'bOk FALSE');
AssertEquals_STRING('type', fb.sParseError, 'sParseError');
TEST_FINISHED();
END_METHOD

METHOD PRIVATE Test_TypeDesconhecido_bOkFalse
VAR
	fb  : FB_DfiPayloadParser;
	cfg : ST_DfiConfig;
END_VAR
TEST('TypeDesconhecido_bOkFalse');
cfg.sTopicEstoque := 'dataflow/estoque';
fb(bExecute := TRUE, sTopic := 'dataflow/estoque',
   sPayload := '{"type":"sensores","pecaA":1,"pecaB":2,"pecaC":3}', stConfig := cfg);
AssertFalse(fb.bOk, 'bOk FALSE');
AssertEquals_STRING('type', fb.sParseError, 'sParseError');
TEST_FINISHED();
END_METHOD

METHOD PRIVATE Test_Estoque_CampoFaltando_bOkFalse
VAR
	fb  : FB_DfiPayloadParser;
	cfg : ST_DfiConfig;
END_VAR
TEST('Estoque_CampoFaltando_bOkFalse');
cfg.sTopicEstoque := 'dataflow/estoque';
fb(bExecute := TRUE, sTopic := 'dataflow/estoque',
   sPayload := '{"type":"estoque","pecaA":1,"pecaB":2}', stConfig := cfg);
AssertFalse(fb.bOk, 'bOk FALSE');
AssertEquals_STRING('campo', fb.sParseError, 'sParseError');
TEST_FINISHED();
END_METHOD

METHOD PRIVATE Test_Estoque_Negativo_bOkFalse
VAR
	fb  : FB_DfiPayloadParser;
	cfg : ST_DfiConfig;
END_VAR
TEST('Estoque_Negativo_bOkFalse');
cfg.sTopicEstoque := 'dataflow/estoque'; cfg.nEstoqueMax := 999;
fb(bExecute := TRUE, sTopic := 'dataflow/estoque',
   sPayload := '{"type":"estoque","pecaA":-1,"pecaB":2,"pecaC":3}', stConfig := cfg);
AssertFalse(fb.bOk, 'bOk FALSE');
AssertEquals_STRING('faixa', fb.sParseError, 'sParseError');
TEST_FINISHED();
END_METHOD

METHOD PRIVATE Test_Estoque_AcimaDoMax_bOkFalse
VAR
	fb  : FB_DfiPayloadParser;
	cfg : ST_DfiConfig;
END_VAR
TEST('Estoque_AcimaDoMax_bOkFalse');
cfg.sTopicEstoque := 'dataflow/estoque'; cfg.nEstoqueMax := 10;
fb(bExecute := TRUE, sTopic := 'dataflow/estoque',
   sPayload := '{"type":"estoque","pecaA":1,"pecaB":2,"pecaC":11}', stConfig := cfg);
AssertFalse(fb.bOk, 'bOk FALSE');
AssertEquals_STRING('faixa', fb.sParseError, 'sParseError');
TEST_FINISHED();
END_METHOD

METHOD PRIVATE Test_Evento_SemCampoEvento_bOkFalse
VAR
	fb  : FB_DfiPayloadParser;
	cfg : ST_DfiConfig;
END_VAR
TEST('Evento_SemCampoEvento_bOkFalse');
cfg.sTopicEventos := 'dataflow/eventos';
fb(bExecute := TRUE, sTopic := 'dataflow/eventos',
   sPayload := '{"type":"evento","peca":"A"}', stConfig := cfg);
AssertFalse(fb.bOk, 'bOk FALSE');
AssertEquals_STRING('campo', fb.sParseError, 'sParseError');
TEST_FINISHED();
END_METHOD

METHOD PRIVATE Test_Evento_PecaInvalida_bOkFalse
VAR
	fb  : FB_DfiPayloadParser;
	cfg : ST_DfiConfig;
END_VAR
TEST('Evento_PecaInvalida_bOkFalse');
cfg.sTopicEventos := 'dataflow/eventos';
fb(bExecute := TRUE, sTopic := 'dataflow/eventos',
   sPayload := '{"type":"evento","evento":"entrega","peca":"D"}', stConfig := cfg);
AssertFalse(fb.bOk, 'bOk FALSE');
AssertEquals_STRING('peca', fb.sParseError, 'sParseError');
TEST_FINISHED();
END_METHOD

METHOD PRIVATE Test_Evento_PecaAusente_Ok_PecaVazia
VAR
	fb  : FB_DfiPayloadParser;
	cfg : ST_DfiConfig;
END_VAR
TEST('Evento_PecaAusente_Ok_PecaVazia');
cfg.sTopicEventos := 'dataflow/eventos';
fb(bExecute := TRUE, sTopic := 'dataflow/eventos',
   sPayload := '{"type":"evento","evento":"inicializacao"}', stConfig := cfg);
AssertTrue(fb.bOk, 'bOk TRUE');
AssertEquals_STRING('', fb.stEvento.sPeca, 'peca vazia');
TEST_FINISHED();
END_METHOD

METHOD PRIVATE Test_Evento_DetalheComAspa_bOkFalse
VAR
	fb  : FB_DfiPayloadParser;
	cfg : ST_DfiConfig;
END_VAR
TEST('Evento_DetalheComAspa_bOkFalse');
cfg.sTopicEventos := 'dataflow/eventos';
fb(bExecute := TRUE, sTopic := 'dataflow/eventos',
   sPayload := '{"type":"evento","evento":"erro","tipo":"ti$'meout","peca":"B"}', stConfig := cfg);
AssertFalse(fb.bOk, 'bOk FALSE');
AssertEquals_STRING('sanit', fb.sParseError, 'sParseError');
TEST_FINISHED();
END_METHOD

METHOD PRIVATE Test_Evento_EventoComPontoEVirgula_bOkFalse
VAR
	fb  : FB_DfiPayloadParser;
	cfg : ST_DfiConfig;
END_VAR
TEST('Evento_EventoComPontoEVirgula_bOkFalse');
cfg.sTopicEventos := 'dataflow/eventos';
fb(bExecute := TRUE, sTopic := 'dataflow/eventos',
   sPayload := '{"type":"evento","evento":"a;b"}', stConfig := cfg);
AssertFalse(fb.bOk, 'bOk FALSE');
AssertEquals_STRING('sanit', fb.sParseError, 'sParseError');
TEST_FINISHED();
END_METHOD

METHOD PRIVATE Test_Evento_DetalheLongo_Truncado
VAR
	fb      : FB_DfiPayloadParser;
	cfg     : ST_DfiConfig;
	sTipo80 : STRING(120);
	sBig    : STRING(510);
	i       : INT;
END_VAR
TEST('Evento_DetalheLongo_Truncado');
cfg.sTopicEventos := 'dataflow/eventos';
sTipo80 := '';
FOR i := 1 TO 80 DO
	sTipo80 := CONCAT(sTipo80, 'x');
END_FOR
sBig := CONCAT('{"type":"evento","evento":"erro","tipo":"', CONCAT(sTipo80, '"}'));
fb(bExecute := TRUE, sTopic := 'dataflow/eventos', sPayload := sBig, stConfig := cfg);
AssertTrue(fb.bOk, 'bOk TRUE');
AssertEquals_INT(63, LEN(fb.stEvento.sDetalhe), 'detalhe truncado a 63');
TEST_FINISHED();
END_METHOD

METHOD PRIVATE Test_Evento_PayloadRaw_Preenchido
VAR
	fb  : FB_DfiPayloadParser;
	cfg : ST_DfiConfig;
END_VAR
TEST('Evento_PayloadRaw_Preenchido');
cfg.sTopicEventos := 'dataflow/eventos';
fb(bExecute := TRUE, sTopic := 'dataflow/eventos',
   sPayload := '{"type":"evento","evento":"entrega","peca":"A"}', stConfig := cfg);
AssertTrue(fb.bOk, 'bOk TRUE');
AssertEquals_STRING('{type:evento,evento:entrega,peca:A}', fb.stEvento.sPayloadRaw, 'payload_raw pos-strip');
AssertTrue(LEN(fb.stEvento.sPayloadRaw) <= 254, 'payload_raw <= 254');
TEST_FINISHED();
END_METHOD

METHOD PRIVATE Test_TopicoDesconhecido_bOkFalse
VAR
	fb  : FB_DfiPayloadParser;
	cfg : ST_DfiConfig;
END_VAR
TEST('TopicoDesconhecido_bOkFalse');
cfg.sTopicEstoque := 'dataflow/estoque';
cfg.sTopicEventos := 'dataflow/eventos';
fb(bExecute := TRUE, sTopic := 'dataflow/sensores',
   sPayload := '{"type":"estoque","pecaA":1,"pecaB":2,"pecaC":3}', stConfig := cfg);
AssertFalse(fb.bOk, 'bOk FALSE');
AssertEquals_STRING('topic', fb.sParseError, 'sParseError');
TEST_FINISHED();
END_METHOD

METHOD PRIVATE Test_StripSqlUnsafe_RemoveAspas
VAR
	sOut : STRING(254);
END_VAR
TEST('StripSqlUnsafe_RemoveAspas');
// entrada: a ' b " c ; d \ e ` f <TAB> g  -> todos os perigosos/controle somem
sOut := F_DfiStripSqlUnsafe('a$'b"c;d\e$60f$09g');
AssertEquals_STRING('abcdefg', sOut, 'strip de aspas / ; / barra / crase / controle');
TEST_FINISHED();
END_METHOD

END_FUNCTION_BLOCK

// ---- POUs/fb/FB_DfiPayloadParser.TcPOU
FUNCTION_BLOCK FB_DfiPayloadParser
VAR_INPUT
	sTopic   : STRING(255);
	sPayload : STRING(510);
	stConfig : ST_DfiConfig;
	bExecute : BOOL;
END_VAR
VAR_OUTPUT
	bDone       : BOOL;
	bOk         : BOOL;
	eKind       : E_DfiRowKind;
	stEstoque   : ST_EstoqueSnapshot;
	stEvento    : ST_EventoDfi;
	sParseError : STRING(120);
END_VAR
VAR
	fbJson    : Tc3_JsonXml.FB_JsonDomParser;
	fbTrig    : R_TRIG;
	jsonRoot  : Tc3_JsonXml.SJsonValue;
	bEstoque  : BOOL;
	bEvento   : BOOL;
	sType     : STRING(63);
	sEv       : STRING(254);
	sEvClean  : STRING(254);
	sPeca     : STRING(254);
	sTipo     : STRING(254);
	sDetClean : STRING(254);
	nMax      : DINT;
	nA        : DINT;
	nB        : DINT;
	nC        : DINT;
	bV        : BOOL;
	bFound    : BOOL;
END_VAR

// Executa somente na borda de subida de bExecute (Step 4).
fbTrig(CLK := bExecute);
IF NOT fbTrig.Q THEN
	RETURN;
END_IF

// 1) limpa saidas
bDone       := FALSE;
bOk         := FALSE;
sParseError := '';
eKind       := E_DfiRowKind.ESTOQUE_MUDANCA;
stEstoque.nA := 0;
stEstoque.nB := 0;
stEstoque.nC := 0;
stEvento.sEvento     := '';
stEvento.sPeca       := '';
stEvento.sDetalhe    := '';
stEvento.sPayloadRaw := '';

// 2) roteamento por topico
bEstoque := (sTopic = stConfig.sTopicEstoque);
bEvento  := (sTopic = stConfig.sTopicEventos);
IF (NOT bEstoque) AND (NOT bEvento) THEN
	sParseError := 'topic';
	bDone := TRUE;
	RETURN;
END_IF

// 3) parse do JSON (ParseDocument retorna a raiz; 0 => documento invalido)
jsonRoot := fbJson.ParseDocument(sPayload);
IF jsonRoot = 0 THEN
	sParseError := 'json';
	bDone := TRUE;
	RETURN;
END_IF

// 4) campo 'type'
sType := THIS^.GetStr(jsonRoot, 'type');
IF (NOT bFound) OR (sType = '') THEN
	sParseError := 'type';
	bDone := TRUE;
	RETURN;
END_IF
IF bEstoque AND (sType <> 'estoque') THEN
	sParseError := 'type';
	bDone := TRUE;
	RETURN;
END_IF
IF bEvento AND (sType <> 'evento') THEN
	sParseError := 'type';
	bDone := TRUE;
	RETURN;
END_IF

// 5) ramo ESTOQUE
IF bEstoque THEN
	nMax := stConfig.nEstoqueMax;
	nA := THIS^.GetInt(jsonRoot, 'pecaA');
	IF NOT bV THEN
		sParseError := 'campo';
		bDone := TRUE;
		RETURN;
	END_IF
	nB := THIS^.GetInt(jsonRoot, 'pecaB');
	IF NOT bV THEN
		sParseError := 'campo';
		bDone := TRUE;
		RETURN;
	END_IF
	nC := THIS^.GetInt(jsonRoot, 'pecaC');
	IF NOT bV THEN
		sParseError := 'campo';
		bDone := TRUE;
		RETURN;
	END_IF
	IF (nA < 0) OR (nA > nMax)
	OR (nB < 0) OR (nB > nMax)
	OR (nC < 0) OR (nC > nMax) THEN
		sParseError := 'faixa';
		bDone := TRUE;
		RETURN;
	END_IF
	stEstoque.nA := DINT_TO_INT(nA);
	stEstoque.nB := DINT_TO_INT(nB);
	stEstoque.nC := DINT_TO_INT(nC);
	eKind := E_DfiRowKind.ESTOQUE_MUDANCA;
	bOk   := TRUE;
	bDone := TRUE;
	RETURN;
END_IF

// 6) ramo EVENTO
sEv := THIS^.GetStr(jsonRoot, 'evento');
IF (NOT bFound) OR (sEv = '') THEN
	sParseError := 'campo';
	bDone := TRUE;
	RETURN;
END_IF
IF NOT F_DfiSanitizeText(sEv, 23) THEN
	sParseError := 'sanit';
	bDone := TRUE;
	RETURN;
END_IF

// peca: se presente precisa ser 'A' | 'B' | 'C'; se ausente => ''
IF THIS^.HasKey(jsonRoot, 'peca') THEN
	sPeca := THIS^.GetStr(jsonRoot, 'peca');
	IF (sPeca <> 'A') AND (sPeca <> 'B') AND (sPeca <> 'C') THEN
		sParseError := 'peca';
		bDone := TRUE;
		RETURN;
	END_IF
	stEvento.sPeca := sPeca;
ELSE
	stEvento.sPeca := '';
END_IF

// tipo -> detalhe: se presente sanitiza (63); se ausente => ''
IF THIS^.HasKey(jsonRoot, 'tipo') THEN
	sTipo := THIS^.GetStr(jsonRoot, 'tipo');
	IF NOT F_DfiSanitizeText(sTipo, 63) THEN
		sParseError := 'sanit';
		bDone := TRUE;
		RETURN;
	END_IF
	stEvento.sDetalhe := sDetClean;
ELSE
	stEvento.sDetalhe := '';
END_IF

// payload_raw: filtro leve, NAO bloqueia a linha (auditoria best-effort)
stEvento.sEvento     := sEvClean;
stEvento.sPayloadRaw := F_DfiStripSqlUnsafe(LEFT(sPayload, 254));
eKind := E_DfiRowKind.EVENTO;
bOk   := TRUE;
bDone := TRUE;

METHOD PRIVATE GetInt : DINT
VAR_INPUT
	dom   : Tc3_JsonXml.SJsonValue;
	sName : STRING(80);
END_VAR
VAR_OUTPUT
	bValid : BOOL;
END_VAR
VAR
	j    : Tc3_JsonXml.SJsonValue;
	lVal : LINT;
END_VAR
// Wrapper isolado sobre a API Tc3_JsonXml.
// bValid = TRUE somente se a chave existe E o valor e um inteiro.
bValid := FALSE;
GetInt := 0;
IF NOT fbJson.HasMember(dom, sName) THEN
	RETURN;
END_IF
j := fbJson.FindMember(dom, sName);
IF j = 0 THEN
	RETURN;
END_IF
IF NOT fbJson.IsInt(j) THEN
	RETURN;
END_IF
lVal := fbJson.GetInt(j);
GetInt := LINT_TO_DINT(lVal);
bValid := TRUE;
END_METHOD

METHOD PRIVATE GetStr : STRING(255)
VAR_INPUT
	dom   : Tc3_JsonXml.SJsonValue;
	sName : STRING(80);
END_VAR
VAR_OUTPUT
	bFound : BOOL;
END_VAR
VAR
	j : Tc3_JsonXml.SJsonValue;
END_VAR
// Wrapper isolado sobre a API Tc3_JsonXml.
// bFound = TRUE somente se a chave existe E o valor e string.
bFound := FALSE;
GetStr := '';
IF NOT fbJson.HasMember(dom, sName) THEN
	RETURN;
END_IF
j := fbJson.FindMember(dom, sName);
IF j = 0 THEN
	RETURN;
END_IF
IF NOT fbJson.IsString(j) THEN
	RETURN;
END_IF
GetStr := fbJson.GetString(j);
bFound := TRUE;
END_METHOD

METHOD PRIVATE HasKey : BOOL
VAR_INPUT
	dom   : Tc3_JsonXml.SJsonValue;
	sName : STRING(80);
END_VAR
// Wrapper isolado sobre a API Tc3_JsonXml (um unico ponto a corrigir no checkpoint).
HasKey := fbJson.HasMember(dom, sName);
END_METHOD

END_FUNCTION_BLOCK

// ---- POUs/fb/F_DfiSanitizeText.TcPOU
FUNCTION F_DfiSanitizeText : BOOL
VAR_INPUT
	sEntrada     : STRING(254);
	nMaxLen : INT;
END_VAR
VAR_OUTPUT
	sOut : STRING(254);
END_VAR
VAR
	i, n : INT;
	c    : BYTE;
	p    : POINTER TO BYTE;
END_VAR

n := LEN(sEntrada);
p := ADR(sEntrada);
FOR i := 0 TO n - 1 DO
	c := p[i];
	IF NOT ( (c >= 65 AND c <= 90)  OR   // A-Z
	         (c >= 97 AND c <= 122) OR   // a-z
	         (c >= 48 AND c <= 57)  OR   // 0-9
	         (c = 32) OR (c = 95) OR (c = 45) ) THEN  // space _ -
		F_DfiSanitizeText := FALSE;
		RETURN;
	END_IF
END_FOR
IF n > nMaxLen THEN
	sOut := LEFT(sEntrada, nMaxLen);
ELSE
	sOut := sEntrada;
END_IF
F_DfiSanitizeText := TRUE;

END_FUNCTION

// ---- POUs/fb/F_DfiStripSqlUnsafe.TcPOU
FUNCTION F_DfiStripSqlUnsafe : STRING(254)
VAR_INPUT
	sEntrada : STRING(254);
END_VAR
VAR
	i, n, k : INT;
	c       : BYTE;
	pIn     : POINTER TO BYTE;
	pOut    : POINTER TO BYTE;
	sRes    : STRING(254);
END_VAR

// Filtro leve para payload_raw (auditoria): copia sIn descartando apenas
// os bytes  39 (')  34 (")  59 (;)  92 (\)  96 (`)  e qualquer byte < 16#20.
// Mantem todo o resto (chaves, dois-pontos, virgulas...). Teto em 254 chars.
// Varredura por ponteiro de bytes, no estilo de F_DfiSanitizeText.
n    := LEN(sEntrada);
pIn  := ADR(sEntrada);
pOut := ADR(sRes);
k    := 0;
FOR i := 0 TO n - 1 DO
	IF k >= 254 THEN
		EXIT;
	END_IF
	c := pIn[i];
	IF NOT ( (c = 39) OR (c = 34) OR (c = 59) OR (c = 92) OR (c = 96) OR (c < 16#20) ) THEN
		pOut[k] := c;
		k := k + 1;
	END_IF
END_FOR
pOut[k] := 0;
F_DfiStripSqlUnsafe := sRes;

END_FUNCTION

// ---- POUs/test/FB_DfiSqlBuilder_Tests.TcPOU
FUNCTION_BLOCK FB_DfiSqlBuilder_Tests EXTENDS TcUnit.FB_TestSuite
VAR
END_VAR

Test_Build_EstoqueMudanca();
Test_Build_EstoquePeriodico_OrigemPeriodico();
Test_Build_Evento_ComPecaEDetalhe();
Test_Build_Evento_SemPeca_SemDetalhe_UsaNULL();
Test_Build_Evento_PayloadLongo_NaoTrunca();

METHOD PRIVATE Test_Build_EstoqueMudanca
VAR
	fb : FB_DfiSqlBuilder;
	linha : ST_DfiRow;
	conjunto : STRING(511);
END_VAR
TEST('Build_EstoqueMudanca');
linha.eKind := E_DfiRowKind.ESTOQUE_MUDANCA;
linha.sTsPlc := '2026-09-08 10:11:12.345';
linha.stEstoque.nA := 4; linha.stEstoque.nB := 5; linha.stEstoque.nC := 6;
fb.Build(linha);
AssertEquals_STRING(
  Expected := 'INSERT INTO estoque_hist (ts_plc,estoque_a,estoque_b,estoque_c,origem) VALUES ($'2026-09-08 10:11:12.345$',4,5,6,$'mudanca$');',
  Actual := conjunto, Message := 'SQL estoque mudanca');
TEST_FINISHED();
END_METHOD

METHOD PRIVATE Test_Build_EstoquePeriodico_OrigemPeriodico
VAR
	fb : FB_DfiSqlBuilder;
	linha : ST_DfiRow;
	conjunto : STRING(511);
END_VAR
TEST('Build_EstoquePeriodico');
linha.eKind := E_DfiRowKind.ESTOQUE_PERIODICO;
linha.sTsPlc := '2026-09-08 10:12:12.000';
linha.stEstoque.nA := 0; linha.stEstoque.nB := 1; linha.stEstoque.nC := 2;
fb.Build(linha);
AssertEquals_STRING(
  Expected := 'INSERT INTO estoque_hist (ts_plc,estoque_a,estoque_b,estoque_c,origem) VALUES ($'2026-09-08 10:12:12.000$',0,1,2,$'periodico$');',
  Actual := conjunto, Message := 'SQL estoque periodico');
TEST_FINISHED();
END_METHOD

METHOD PRIVATE Test_Build_Evento_ComPecaEDetalhe
VAR
	fb : FB_DfiSqlBuilder;
	linha : ST_DfiRow;
	conjunto : STRING(511);
END_VAR
TEST('Build_Evento_ComPecaEDetalhe');
linha.eKind := E_DfiRowKind.EVENTO;
linha.sTsPlc := '2026-09-08 10:13:00.000';
linha.stEvento.sEvento := 'erro'; linha.stEvento.sPeca := 'B'; linha.stEvento.sDetalhe := 'timeout';
linha.stEvento.sPayloadRaw := '{type:evento,evento:erro}';
fb.Build(linha);
AssertEquals_STRING(
  Expected := 'INSERT INTO eventos_hist (ts_plc,evento,peca,detalhe,payload_raw) VALUES ($'2026-09-08 10:13:00.000$',$'erro$',$'B$',$'timeout$',$'{type:evento,evento:erro}$');',
  Actual := conjunto, Message := 'SQL evento completo');
TEST_FINISHED();
END_METHOD

METHOD PRIVATE Test_Build_Evento_PayloadLongo_NaoTrunca
VAR
	fb    : FB_DfiSqlBuilder;
	linha : ST_DfiRow;
	conjunto     : STRING(511);
	sBig  : STRING(254);
	sDet  : STRING(63);
	nLen  : UINT;
	bRet  : BOOL;
	pB    : POINTER TO BYTE;
	i     : INT;
END_VAR
TEST('Build_Evento_PayloadLongo_NaoTrunca');

// payload_raw no limite: 254 'x' (STRING(254)); 254 < 255 -> CONCAT ok aqui
sBig := '';
FOR i := 1 TO 254 DO
	sBig := CONCAT(sBig, 'x');
END_FOR

// detalhe no limite: 63 'y' (STRING(63))
sDet := '';
FOR i := 1 TO 63 DO
	sDet := CONCAT(sDet, 'y');
END_FOR

linha.eKind := E_DfiRowKind.EVENTO;
linha.sTsPlc := '2026-09-08 10:15:00.000';
linha.stEvento.sEvento := 'entrega';
linha.stEvento.sPeca := 'C';
linha.stEvento.sDetalhe := sDet;
linha.stEvento.sPayloadRaw := sBig;

bRet := fb.Build(stRow := linha, sCmd => conjunto, nCmdLen => nLen);

// prefixo decodificado = "INSERT INTO eventos_hist (ts_plc,evento,peca,detalhe,payload_raw) VALUES (
//   '2026-09-08 10:15:00.000','entrega','C','<63 y>','"  -> 181 bytes
// + payload 254 + "');" 3  -> 438 bytes (sem terminador)
AssertTrue(bRet, 'Build retornou TRUE para payload longo');
AssertEquals_UINT(Expected := 438, Actual := nLen, Message := 'comprimento total sem truncar');

// cauda intacta: ...x  '  )  ;
pB := ADR(conjunto);
AssertTrue(pB[nLen - 1] = 16#3B, 'ultimo byte = ; (0x3B)');
AssertTrue(pB[nLen - 2] = 16#29, 'penultimo byte = ) (0x29)');
AssertTrue(pB[nLen - 3] = 16#27, 'antepenultimo byte = aspa (0x27)');
AssertTrue(pB[nLen - 4] = 16#78, 'ultimo char do payload = x (0x78)');

TEST_FINISHED();
END_METHOD

METHOD PRIVATE Test_Build_Evento_SemPeca_SemDetalhe_UsaNULL
VAR
	fb : FB_DfiSqlBuilder;
	linha : ST_DfiRow;
	conjunto : STRING(511);
END_VAR
TEST('Build_Evento_SemPeca_UsaNULL');
linha.eKind := E_DfiRowKind.EVENTO;
linha.sTsPlc := '2026-09-08 10:14:00.000';
linha.stEvento.sEvento := 'inicializacao'; linha.stEvento.sPeca := ''; linha.stEvento.sDetalhe := '';
linha.stEvento.sPayloadRaw := '';
fb.Build(linha);
AssertEquals_STRING(
  Expected := 'INSERT INTO eventos_hist (ts_plc,evento,peca,detalhe,payload_raw) VALUES ($'2026-09-08 10:14:00.000$',$'inicializacao$',NULL,NULL,$'$');',
  Actual := conjunto, Message := 'peca/detalhe NULL, payload_raw string vazia');
TEST_FINISHED();
END_METHOD

END_FUNCTION_BLOCK

// ---- POUs/fb/FB_DfiSqlBuilder.TcPOU
FUNCTION_BLOCK FB_DfiSqlBuilder
VAR
	fbFmt   : Tc2_Utilities.FB_FormatString;
	sOrigem : STRING(80);
	sPeca   : STRING(80);
	sDet    : STRING(80);
END_VAR

// Sem logica no corpo: a construcao do INSERT e feita pelo metodo Build.

METHOD Build : BOOL
VAR_INPUT
	stRow : ST_DfiRow;
END_VAR
VAR_OUTPUT
	sCmd    : STRING(511);
	nCmdLen : UINT;         // comprimento em bytes de sCmd (sem o terminador), setado em todo caminho
END_VAR
VAR
	sPrefix : STRING(255);  // prefixo fixo+curto do INSERT de eventos (pior caso ~200 bytes)
	pDst    : POINTER TO BYTE;
	pPre    : POINTER TO BYTE;
	pPay    : POINTER TO BYTE;
	nP      : DINT;
	nPay    : DINT;
	i       : DINT;
END_VAR
// Gera o comando INSERT exato para o tipo de linha (stRow.eKind).
// Escape de aspa simples em literal ST do TwinCAT: $'  (nao '').
// eventos: o statement de pior caso (~454 bytes) NAO cabe em STRING(255).
// FB_FormatString/CONCAT/LEFT/... sao todos limitados a T_MaxString, entao o
// payload nunca passa por eles: FB_FormatString monta so o prefixo curto e o
// restante e montado por ponteiro de bytes direto em sCmd (STRING(511)),
// no estilo de F_DfiStripSqlUnsafe.
sCmd    := '';
nCmdLen := 0;

CASE stRow.eKind OF

	E_DfiRowKind.ESTOQUE_MUDANCA, E_DfiRowKind.ESTOQUE_PERIODICO:
		// SEL(G, IN0, IN1): G=FALSE -> IN0 ; G=TRUE -> IN1
		// eKind = ESTOQUE_MUDANCA   -> 'mudanca'
		// eKind = ESTOQUE_PERIODICO -> 'periodico'
		sOrigem := SEL(stRow.eKind = E_DfiRowKind.ESTOQUE_MUDANCA, 'periodico', 'mudanca');
		fbFmt(
			sFormat := 'INSERT INTO estoque_hist (ts_plc,estoque_a,estoque_b,estoque_c,origem) VALUES ($'%s$',%d,%d,%d,$'%s$');',
			arg1 := Tc2_Utilities.F_String(stRow.sTsPlc),
			arg2 := Tc2_Utilities.F_INT(stRow.stEstoque.nA),
			arg3 := Tc2_Utilities.F_INT(stRow.stEstoque.nB),
			arg4 := Tc2_Utilities.F_INT(stRow.stEstoque.nC),
			arg5 := Tc2_Utilities.F_String(sOrigem),
			sOut => sCmd);
		// comprimento em bytes de sCmd (stdlib nao mede > 255): varre ate o 0
		pPre := ADR(sCmd);
		nP := 0;
		WHILE (nP < 511) AND (pPre[nP] <> 0) DO
			nP := nP + 1;
		END_WHILE
		nCmdLen := DINT_TO_UINT(nP);
		Build := NOT fbFmt.bError;

	E_DfiRowKind.EVENTO:
		// peca / detalhe: string entre aspas quando presente, senao literal NULL
		IF stRow.stEvento.sPeca = '' THEN
			sPeca := 'NULL';
		ELSE
			sPeca := CONCAT('$'', CONCAT(stRow.stEvento.sPeca, '$''));
		END_IF

		IF stRow.stEvento.sDetalhe = '' THEN
			sDet := 'NULL';
		ELSE
			sDet := CONCAT('$'', CONCAT(stRow.stEvento.sDetalhe, '$''));
		END_IF

		// prefixo fixo+curto: termina com a aspa de abertura de payload_raw
		// e NADA depois (o proprio payload e o fecho vem por ponteiro).
		fbFmt(
			sFormat := 'INSERT INTO eventos_hist (ts_plc,evento,peca,detalhe,payload_raw) VALUES ($'%s$',$'%s$',%s,%s,$'',
			arg1 := F_String(stRow.sTsPlc),
			arg2 := F_String(stRow.stEvento.sEvento),
			arg3 := F_String(sPeca),
			arg4 := F_String(sDet),
			sOut => sPrefix);

		IF fbFmt.bError THEN
			Build := FALSE;
			RETURN;
		END_IF

		// comprimento do prefixo (varre ADR(sPrefix) ate o 0)
		pPre := ADR(sPrefix);
		nP := 0;
		WHILE (nP < 255) AND (pPre[nP] <> 0) DO
			nP := nP + 1;
		END_WHILE

		// comprimento do payload bruto (varre ate o 0, teto 254)
		pPay := ADR(stRow.stEvento.sPayloadRaw);
		nPay := 0;
		WHILE (nPay < 254) AND (pPay[nPay] <> 0) DO
			nPay := nPay + 1;
		END_WHILE

		// guarda de buffer: sCmd e STRING(511) -> no maximo 510 bytes de dados
		IF (nP + nPay + 3) > 510 THEN
			sCmd    := '';
			nCmdLen := 0;
			Build   := FALSE;
			RETURN;
		END_IF

		// montagem por ponteiro: prefixo + payload + fecha aspa/paren/;  + NUL
		pDst := ADR(sCmd);

		FOR i := 0 TO nP - 1 DO
			pDst[i] := pPre[i];
		END_FOR

		FOR i := 0 TO nPay - 1 DO
			pDst[nP + i] := pPay[i];
		END_FOR

		pDst[nP + nPay + 0] := 16#27;   // aspa simples '
		pDst[nP + nPay + 1] := 16#29;   // parentese )
		pDst[nP + nPay + 2] := 16#3B;   // ponto-e-virgula ;
		pDst[nP + nPay + 3] := 0;       // terminador NUL

		nCmdLen := DINT_TO_UINT(nP + nPay + 3);
		Build   := TRUE;

ELSE
	sCmd    := '';
	nCmdLen := 0;
	Build   := FALSE;

END_CASE
END_METHOD

END_FUNCTION_BLOCK

// ---- POUs/test/F_DfiNowString_Tests.TcPOU
FUNCTION_BLOCK F_DfiNowString_Tests EXTENDS TcUnit.FB_TestSuite
VAR
END_VAR

Test_Formato_23Chars_ComSeparadores();

METHOD PRIVATE Test_Formato_23Chars_ComSeparadores
VAR
	conjunto: STRING(23);
	i       : INT;
	c       : STRING(1);
	bDigito : BOOL;
END_VAR
TEST('Formato_23Chars');
conjunto := F_DfiNowString();
AssertEquals_INT(23, LEN(conjunto), 'comprimento 23');
AssertEquals_STRING('-', MID(conjunto, 1, 5), 'traco em pos 5');
AssertEquals_STRING('-', MID(conjunto, 1, 8), 'traco em pos 8');
AssertEquals_STRING(' ', MID(conjunto, 1, 11), 'espaco em pos 11');
AssertEquals_STRING(':', MID(conjunto, 1, 14), 'dois-pontos pos 14');
AssertEquals_STRING('.', MID(conjunto, 1, 20), 'ponto pos 20');
// separador extra de minutos e checagem de digitos nas posicoes numericas
AssertEquals_STRING(':', MID(conjunto, 1, 17), 'dois-pontos pos 17');
bDigito := TRUE;
FOR i := 1 TO 23 DO
	IF i <> 5 AND i <> 8 AND i <> 11 AND i <> 14 AND i <> 17 AND i <> 20 THEN
		c := MID(conjunto, 1, i);
		IF (c < '0') OR (c > '9') THEN
			bDigito := FALSE;
		END_IF
	END_IF
END_FOR
AssertTrue(bDigito, 'campos numericos sao digitos 0-9');
TEST_FINISHED();
END_METHOD

END_FUNCTION_BLOCK

// ---- POUs/test/FB_DfiDbWriter_Tests.TcPOU
FUNCTION_BLOCK FB_DfiDbWriter_Tests EXTENDS TcUnit.FB_TestSuite
VAR
END_VAR
VAR CONSTANT
	// Espelham as constantes de FB_DfiDbWriter_Fake (VAR CONSTANT de FB nao e
	// visivel de fora da instancia). Manter os dois blocos em sincronia.
	SCRIPT_OK         : INT := 1;
	SCRIPT_EXEC_ERROR : INT := 2;
	SCRIPT_DB_LOST    : INT := 3;
END_VAR

Test_Sucesso_PopEContagem();
Test_ErroExecute_NaoPop_BackoffCresce();
Test_DbLost_DuranteExecute_VoltaIdle_SemPerder();
Test_PeriodicoTambemAtualizaBaseline();

METHOD PRIVATE Test_DbLost_DuranteExecute_VoltaIdle_SemPerder
VAR
	fbBuf : FB_DfiRowBuffer := (nCapacity := 8);
	sut   : FB_DfiDbWriter_Fake;
	cfg   : ST_DfiConfig;
	linha     : ST_DfiRow;
	i     : INT;
END_VAR
TEST('DbLost_SemPerder');
sut.SetScript(SCRIPT_DB_LOST);
fbBuf.Push(linha);
FOR i := 1 TO 20 DO sut(stConfig := cfg, fbBuffer := fbBuf); END_FOR
AssertEquals_UDINT(1, fbBuf.nCount, 'linha preservada em DB_LOST');
TEST_FINISHED();
END_METHOD

METHOD PRIVATE Test_ErroExecute_NaoPop_BackoffCresce
VAR
	fbBuf : FB_DfiRowBuffer := (nCapacity := 8);
	sut   : FB_DfiDbWriter_Fake;
	cfg   : ST_DfiConfig;
	linha     : ST_DfiRow;
	i     : INT;
END_VAR
TEST('ErroExecute_NaoPop');
sut.SetScript(SCRIPT_EXEC_ERROR);   // DoExecute retorna 2 (erro)
fbBuf.Push(linha);
FOR i := 1 TO 30 DO sut(stConfig := cfg, fbBuffer := fbBuf); END_FOR
AssertEquals_UDINT(1, fbBuf.nCount, 'linha PRESERVADA apos erro');
AssertTrue(sut.nErrors >= 1, 'nErrors incrementa');
AssertTrue(sut.eState = E_DfiWriterState.ERROR OR sut.eState = E_DfiWriterState.IDLE, 'em ERROR/backoff ou voltando');
TEST_FINISHED();
END_METHOD

METHOD PRIVATE Test_PeriodicoTambemAtualizaBaseline
VAR
	fbBuf : FB_DfiRowBuffer := (nCapacity := 8);
	sut   : FB_DfiDbWriter_Fake;
	cfg   : ST_DfiConfig; linha : ST_DfiRow; i : INT;
END_VAR
TEST('PeriodicoAtualizaBaseline');
sut.SetScript(SCRIPT_OK);
linha.eKind := E_DfiRowKind.ESTOQUE_PERIODICO; linha.stEstoque.nB := 2;
fbBuf.Push(linha);
FOR i := 1 TO 20 DO sut(stConfig := cfg, fbBuffer := fbBuf); END_FOR
AssertTrue(sut.bUltimoGravadoValido, 'baseline valido apos periodico');
AssertEquals_INT(2, sut.stUltimoGravado.nB, 'baseline B=2');
TEST_FINISHED();
END_METHOD

METHOD PRIVATE Test_Sucesso_PopEContagem
VAR
	fbBuf : FB_DfiRowBuffer := (nCapacity := 8);
	sut   : FB_DfiDbWriter_Fake;   // DoExecute sempre retorna 1 (ok) apos 1 ciclo "busy"
	cfg   : ST_DfiConfig;
	linha : ST_DfiRow;
	i     : INT;
END_VAR
TEST('Sucesso_PopEContagem');
sut.SetScript(SCRIPT_OK);      // helper do fake
linha.eKind := E_DfiRowKind.ESTOQUE_MUDANCA; linha.stEstoque.nA := 9;
fbBuf.Push(linha);
FOR i := 1 TO 20 DO sut(stConfig := cfg, fbBuffer := fbBuf); END_FOR
AssertEquals_UDINT(0, fbBuf.nCount, 'linha removida apos sucesso');
AssertEquals_ULINT(1, sut.nRowsWritten, 'nRowsWritten=1');
AssertTrue(sut.bUltimoGravadoValido, 'dedupe baseline valido');
AssertEquals_INT(9, sut.stUltimoGravado.nA, 'dedupe baseline = ultima linha de estoque');
TEST_FINISHED();
END_METHOD

END_FUNCTION_BLOCK

// ---- POUs/test/FB_DfiDbWriter_Fake.TcPOU
// Dublê de teste de FB_DfiDbWriter: sobrescreve apenas o seam DoExecute,
// deixando toda a maquina de estados da classe base rodar de verdade.
// FB_SQLCommandEvt/FB_SQLDatabaseEvt exigem um TwinCAT Database Server real,
// por isso o caminho de banco nao e coberto aqui (bancada, Task 15).
FUNCTION_BLOCK FB_DfiDbWriter_Fake EXTENDS FB_DfiDbWriter
VAR
	nScript    : INT;
	nExecCycle : INT;
END_VAR
VAR CONSTANT
	// Espelhadas em FB_DfiDbWriter_Tests (VAR CONSTANT de FB nao e visivel de
	// fora da instancia). Manter os dois blocos em sincronia.
	SCRIPT_OK         : INT := 1;
	SCRIPT_EXEC_ERROR : INT := 2;
	SCRIPT_DB_LOST    : INT := 3;
END_VAR

// A maquina de estados da base vive no metodo herdado Cycle() (nao
// sobrescrito). Chamado aqui em vez de SUPER^() porque VAR_IN_OUT (fbBuffer)
// nao pode ser religado num SUPER^(). DoExecute/DoConnect continuam
// despachando para os overrides deste fake.
Cycle();

METHOD SetScript
VAR_INPUT
	n : INT;
END_VAR
nScript    := n;
nExecCycle := 0;
// Pula o estado CONNECT: os testes exercitam BUILD/EXECUTE/COMMIT direto.
bDbConnected := TRUE;
eState       := E_DfiWriterState.IDLE;
END_METHOD

METHOD PROTECTED DoConnect : INT
// O fake nunca fala com um banco real: conecta instantaneamente.
// 0 = ocupado, 1 = conectado e comando criado, 2 = erro (mesmo contrato da base).
DoConnect := 1;
END_METHOD

METHOD PROTECTED DoExecute : INT
// 0 = ocupado, 1 = ok, 2 = erro (mesmo contrato do metodo sobrescrito).
IF nScript = SCRIPT_EXEC_ERROR THEN
	DoExecute := 2;

ELSIF nScript = SCRIPT_DB_LOST THEN
	// conexao cai no meio do Execute: a base deve ir para DB_LOST sem Pop
	bDbConnected := FALSE;
	DoExecute := 0;

ELSIF nScript = SCRIPT_OK THEN
	// 1 ciclo "ocupado" e depois sucesso, para exercitar a espera em EXECUTE
	IF nExecCycle = 0 THEN
		nExecCycle := 1;
		DoExecute := 0;
	ELSE
		DoExecute := 1;
	END_IF

ELSE
	DoExecute := 1;
END_IF
END_METHOD

END_FUNCTION_BLOCK

// ---- POUs/fb/FB_DfiDbWriter.TcPOU
FUNCTION_BLOCK FB_DfiDbWriter
VAR_INPUT
	stConfig : ST_DfiConfig;
END_VAR
VAR_IN_OUT
	fbBuffer : FB_DfiRowBuffer;
END_VAR
VAR_OUTPUT
	eState               : E_DfiWriterState;
	bDbConnected         : BOOL;
	nRowsWritten         : ULINT;
	nErrors              : ULINT;
	sLastError           : STRING(255);
	stUltimoGravado      : ST_EstoqueSnapshot;
	bUltimoGravadoValido : BOOL;
END_VAR
VAR
	fbDb      : FB_SQLDatabaseEvt;
	fbCmd     : FB_SQLCommandEvt;
	fbBuild   : FB_DfiSqlBuilder;
	fbBackoff : TON;
	tBackoff  : TIME := T#2S;
	sCmd      : STRING(511);
	nCmdLen   : UINT;
	stRow     : ST_DfiRow;
	stEvt     : Tc3_EventLogger.I_TcMessage;
	nExecRes  : INT;      // ultimo retorno de DoExecute (0=ocupado, 1=ok, 2=erro)
	nConnRes  : INT;      // ultimo retorno de DoConnect (0=ocupado, 1=ok, 2=erro)
	bConnDone : BOOL;     // Connect ja concluiu; falta so ciclar CreateCmd
	bErrCounted : BOOL;   // nErrors ja contabilizado nesta entrada em ERROR
END_VAR

// Maquina de estados de gravacao no banco via TF6420 (spec 4.4).
// Ordem obrigatoria por linha: Peek -> Build -> Execute -> Pop.
// Pop acontece SOMENTE em COMMIT (INSERT sem erro) ou no descarte de uma
// linha envenenada em BUILD (SQL impossivel de montar). Erro de banco,
// timeout ou queda de conexao NUNCA removem a linha: ela fica no buffer.

CASE eState OF

E_DfiWriterState.IDLE:
	IF fbBuffer.nCount > 0 THEN
		IF bDbConnected THEN
			eState := E_DfiWriterState.BUILD;
		ELSE
			eState := E_DfiWriterState.CONNECT;
		END_IF
	END_IF

E_DfiWriterState.CONNECT:
	// DoConnect e o segundo ponto de teste (PROTECTED, sobrescrito pelo fake).
	nConnRes := DoConnect();
	CASE nConnRes OF
	0:
		;   // aguarda: Connect/CreateCmd ainda ciclando
	1:
		bDbConnected := TRUE;
		eState := E_DfiWriterState.BUILD;
	2:
		eState := E_DfiWriterState.ERROR;
	END_CASE

E_DfiWriterState.BUILD:
	IF fbBuffer.Peek() THEN
		IF fbBuild.Build(stRow := stRow, sCmd => sCmd, nCmdLen => nCmdLen) THEN
			eState := E_DfiWriterState.EXECUTE;
		ELSE
			// linha envenenada: nunca vai gerar SQL valido. Descarta para nao
			// travar a fila atras dela, mas contabiliza como erro.
			sLastError := 'sql_build_failed';
			nErrors := nErrors + 1;
			fbBuffer.Pop();
			IF fbBuffer.nCount = 0 THEN
				eState := E_DfiWriterState.IDLE;
			END_IF
		END_IF
	ELSE
		eState := E_DfiWriterState.IDLE;
	END_IF

E_DfiWriterState.EXECUTE:
	// DoExecute e o ponto de teste (PROTECTED, sobrescrito pelo fake nos testes).
	nExecRes := DoExecute();
	IF NOT bDbConnected THEN
		// a conexao caiu durante o Execute: sai sem Pop, linha preservada
		eState := E_DfiWriterState.DB_LOST;
	ELSIF nExecRes = 1 THEN
		eState := E_DfiWriterState.COMMIT;
	ELSIF nExecRes = 2 THEN
		stEvt := fbCmd.ipTcResult;
		eState := E_DfiWriterState.ERROR;
	END_IF
	// nExecRes = 0 -> Execute ainda ciclando, permanece em EXECUTE

E_DfiWriterState.COMMIT:
	fbBuffer.Pop();
	nRowsWritten := nRowsWritten + 1;
	IF (stRow.eKind = E_DfiRowKind.ESTOQUE_MUDANCA) OR (stRow.eKind = E_DfiRowKind.ESTOQUE_PERIODICO) THEN
		// baseline de dedupe so avanca depois que a linha esta gravada de fato
		stUltimoGravado := stRow.stEstoque;
		bUltimoGravadoValido := TRUE;
	END_IF
	tBackoff := T#2S;   // sucesso zera o backoff exponencial
	sLastError := '';   // limpa texto de erro antigo apos gravacao bem sucedida
	IF fbBuffer.nCount = 0 THEN
		eState := E_DfiWriterState.IDLE;
	ELSE
		eState := E_DfiWriterState.BUILD;
	END_IF

E_DfiWriterState.ERROR:
	// conta o erro uma unica vez por entrada no estado (nao a cada ciclo de backoff)
	IF NOT bErrCounted THEN
		nErrors := nErrors + 1;
		bErrCounted := TRUE;
	END_IF
	// RequestEventText pode precisar de varios ciclos; stEvt pode ser NULL quando
	// o erro nao veio do TF6420 (ex.: fake de teste) -> guarda obrigatoria.
	IF stEvt <> 0 THEN
		stEvt.RequestEventText(1033, sLastError, SIZEOF(sLastError));
	END_IF
	fbBackoff(IN := TRUE, PT := tBackoff);
	IF fbBackoff.Q THEN
		fbBackoff(IN := FALSE);
		// SEL(G, IN0, IN1): G=FALSE -> IN0. Dobra o backoff e satura em 30s.
		tBackoff := SEL((tBackoff + tBackoff) > T#30S, tBackoff + tBackoff, T#30S);
		bErrCounted := FALSE;
		// Qualquer erro do TF6420 pode ter deixado a sessao/comando invalidos.
		// Derruba a conexao e limpa os flags para que IDLE -> CONNECT refaca
		// Connect + CreateCmd do zero (fire-and-forget: CONNECT reestabelece tudo).
		fbDb.Disconnect();
		bDbConnected := FALSE;
		bConnDone := FALSE;
		eState := E_DfiWriterState.IDLE;
	END_IF

E_DfiWriterState.DB_LOST:
	// buffer mantem todas as linhas; IDLE reabre a conexao no proximo ciclo
	bDbConnected := FALSE;
	bConnDone := FALSE;
	eState := E_DfiWriterState.IDLE;

ELSE
	// estado invalido (nao deve ocorrer): volta ao repouso
	eState := E_DfiWriterState.IDLE;

END_CASE

METHOD PROTECTED DoConnect : INT
// Seam de teste: retorna 0 = ocupado, 1 = conectado e comando criado, 2 = erro.
// Duas fases cicladas (mesmo idioma de EscreverDB.TcPOU, estados 1 e 2):
// Connect ate retornar TRUE, so entao CreateCmd ate retornar TRUE.
// bConnDone evita re-chamar Connect enquanto CreateCmd ainda cicla.
DoConnect := 0;

IF NOT bConnDone THEN
	IF fbDb.Connect(hDBID := stConfig.nDbId) THEN
		IF fbDb.bError THEN
			stEvt := fbDb.ipTcResult;
			DoConnect := 2;
		ELSE
			bConnDone := TRUE;
		END_IF
	END_IF
ELSE
	IF fbDb.CreateCmd(ADR(fbCmd)) THEN
		bConnDone := FALSE;
		IF fbDb.bError THEN
			stEvt := fbDb.ipTcResult;
			DoConnect := 2;
		ELSE
			DoConnect := 1;
		END_IF
	END_IF
END_IF
END_METHOD

METHOD PROTECTED DoExecute : INT
// Seam de teste: retorna 0 = ocupado, 1 = ok, 2 = erro.
// FB_SQLCommandEvt.Execute e ciclico: retorna TRUE quando a operacao termina.
// cbSQLCmd usa nCmdLen (comprimento real montado por FB_DfiSqlBuilder) e NAO
// SIZEOF(sCmd): o buffer de 512 bytes e quase sempre maior que o comando.
IF fbCmd.Execute(pSQLCmd := ADR(sCmd), cbSQLCmd := UINT_TO_UDINT(nCmdLen)) THEN
	IF fbCmd.bError THEN
		DoExecute := 2;
	ELSE
		DoExecute := 1;
	END_IF
ELSE
	DoExecute := 0;
END_IF
END_METHOD

END_FUNCTION_BLOCK

// ---- POUs/fb/FB_DfiConfigLoader.TcPOU
FUNCTION_BLOCK FB_DfiConfigLoader
VAR_INPUT
	bExecute : BOOL;
	sPath    : STRING(255) := '/etc/dfi/historian.conf';
END_VAR
VAR_OUTPUT
	bDone  : BOOL;
	bError : BOOL;
	stCfg  : ST_DfiConfig;
	sError : STRING(120);
END_VAR
VAR
	fbTrig  : R_TRIG;
	fbParse : FB_DfiCfgParse;
	fbOpen  : Tc2_System.FB_FileOpen;
	fbGets  : Tc2_System.FB_FileGets;
	fbClose : Tc2_System.FB_FileClose;
	nState  : INT;
	hFile   : UINT;
	sText   : STRING(4095);
	sLineBuf : STRING(255);
	bAny    : BOOL;
	nTextLen : INT;
	nAdd    : INT;
	k       : INT;
	pTxt    : POINTER TO BYTE;
	pLine   : POINTER TO BYTE;
	stCfgDefaults : ST_DfiConfig;
END_VAR

// Máquina de estados: abre historian.conf, lê linha a linha para sText,
// fecha o arquivo e entrega o texto a FB_DfiCfgParse.ParseText.
// O handle é sempre fechado (sucesso OU erro).
//
// Nota de API (Tc2_System): membros usados conforme documentação Beckhoff -
//   FB_FileOpen : sPathName, nMode, bExecute, bBusy, bError, nErrId, hFile
//   FB_FileGets : hFile, pBuffer, cbBuffer, bExecute, bBusy, bError, nErrId, bEOF
//   FB_FileClose: hFile, bExecute, bBusy, bError, nErrId
// FB_FileGets grava a linha (sem o terminador) no buffer apontado por pBuffer.

fbTrig(CLK := bExecute);
IF fbTrig.Q AND (nState = 0) THEN
	bDone  := FALSE;
	bError := FALSE;
	sError := '';
	sText  := '';
	sLineBuf := '';
	hFile  := 0;
	bAny   := FALSE;
	nTextLen := 0;
	stCfg  := stCfgDefaults;   // limpa saída: 2ª carga de um .conf que removeu uma chave não mantém o valor anterior
	nState := 10;
END_IF

CASE nState OF

	0: // IDLE
		;

	10: // OPEN
		fbOpen(
			bExecute  := TRUE,
			sPathName := sPath,
			nMode     := Tc2_System.FOPEN_MODEREAD OR Tc2_System.FOPEN_MODETEXT);
		IF NOT fbOpen.bBusy THEN
			IF fbOpen.bError THEN
				sError := 'open';
				bError := TRUE;
				nState := 90;
			ELSE
				hFile  := fbOpen.hFile;
				nState := 20;
			END_IF
			fbOpen(bExecute := FALSE);
		END_IF

	20: // READ (uma linha por ciclo, acumula em sText separando por $N)
		fbGets(
			bExecute := TRUE,
			hFile    := hFile);
		IF NOT fbGets.bBusy THEN
			IF fbGets.bError THEN
				sError := 'read';
				bError := TRUE;
				fbGets(bExecute := FALSE);
				nState := 30;
			ELSIF fbGets.bEOF THEN
				fbGets(bExecute := FALSE);
				nState := 30;
			ELSE
				// Acumula a linha em sText separando por $N, via cópia de bytes
				// (CONCAT/LEN do Tc2_Standard operam em STRING(255) e truncariam
				// sText, que é STRING(4095)).
				pTxt  := ADR(sText);
				pLine := ADR(sLineBuf);
				nAdd  := 0;
				WHILE (nAdd < 255) AND (pLine[nAdd] <> 0) DO
					nAdd := nAdd + 1;
				END_WHILE
				IF bAny AND (nTextLen < 4094) THEN
					pTxt[nTextLen] := 16#0A;   // $N
					nTextLen := nTextLen + 1;
				END_IF
				FOR k := 0 TO nAdd - 1 DO
					IF nTextLen < 4094 THEN
						pTxt[nTextLen] := pLine[k];
						nTextLen := nTextLen + 1;
					END_IF
				END_FOR
				pTxt[nTextLen] := 0;           // NUL-termina sText
				bAny  := TRUE;
				fbGets(bExecute := FALSE);
				IF nTextLen > 4000 THEN
					sError := 'file too big';
					bError := TRUE;
					nState := 30;
				END_IF
				// senão permanece em 20 para ler a próxima linha
			END_IF
		END_IF

	30: // CLOSE (caminho normal e caminho de erro passam por aqui)
		fbClose(bExecute := TRUE, hFile := hFile);
		IF NOT fbClose.bBusy THEN
			fbClose(bExecute := FALSE);
			hFile := 0;
			IF bError THEN
				nState := 90;
			ELSE
				nState := 40;
			END_IF
		END_IF

	40: // PARSE
		fbParse.ParseText(sText, stCfg);
		IF NOT stCfg.bValid THEN
			sError := 'parse/host';
			bError := TRUE;
		END_IF
		bDone  := TRUE;
		nState := 0;

	90: // ERR - garante o arquivo fechado
		IF hFile <> 0 THEN
			fbClose(bExecute := TRUE, hFile := hFile);
			IF NOT fbClose.bBusy THEN
				fbClose(bExecute := FALSE);
				hFile := 0;
			END_IF
		END_IF
		IF hFile = 0 THEN
			bDone  := TRUE;
			nState := 0;
		END_IF

END_CASE

END_FUNCTION_BLOCK

// ---- POUs/fb/FB_DfiMqttSubscriber.TcPOU
FUNCTION_BLOCK FB_DfiMqttSubscriber
VAR_INPUT
	stConfig : ST_DfiConfig;
	bEnable  : BOOL;
END_VAR
VAR_OUTPUT
	bConnected      : BOOL;
	bNewMessage     : BOOL;      // pulso de 1 ciclo quando sTopic/sPayload sao validos
	sTopic          : STRING(255);
	sPayload        : STRING(510);
	nReconnectCount : UDINT;
END_VAR
VAR
	fbMqtt      : FB_IotMqttClient;
	fbMsgQueue  : Tc3_IotBase.FB_IotMqttMessageQueue;   // fila de entrada: precisa ser instanciada
	                                                     // e conectada em fbMqtt.ipMessageQueue -
	                                                     // o client NAO cria isso sozinho (confirmado
	                                                     // contra infosys.beckhoff.com/.../3391755403.html
	                                                     // apos ipMessageQueue ficar 0 em bancada real)
	fbMessage   : Tc3_IotBase.FB_IotMqttMessage;
	bParamsSet    : BOOL;
	bWasConnected : BOOL;
	bSubEstoque, bSubEventos : BOOL;
END_VAR

// TF6701 API - confirmado contra infosys.beckhoff.com/.../tf6701_tc3_iot_communication_mqtt
// apos bug real em bancada (ipMessageQueue chegava sempre 0 - ver historico do FB_init):
//   FB_IotMqttClient.sHostName            : STRING  -> host do broker
//   FB_IotMqttClient.nHostPort            : UINT    -> porta do broker
//   FB_IotMqttClient.sClientId            : STRING  -> id fixo do cliente
//   FB_IotMqttClient.stMQTT.sUserName     : STRING  -> usuario (pode ser .sUsername)  [ApplyBrokerParams]
//   FB_IotMqttClient.stMQTT.sUserPassword : STRING  -> senha                          [ApplyBrokerParams]
//   FB_IotMqttClient.stTLS.sCA            : STRING  -> caminho do CA PEM              [ApplyBrokerParams]
//   FB_IotMqttClient.ipMessageQueue       : I_IotMqttMessageQueue  -> ENTRADA; o client
//       NAO cria a fila sozinho. Precisa de uma FB_IotMqttMessageQueue propria (fbMsgQueue)
//       atribuida ANTES do 1o Execute()                                              [ApplyBrokerParams]
//   FB_IotMqttClient.Execute(bConnect := BOOL) : BOOL  -> chamada ciclica de conexao
//   FB_IotMqttClient.bConnected           : BOOL    -> estado atual da conexao
//   FB_IotMqttClient.Subscribe(sTopic := STRING, eQoS := Tc3_IotBase.TcIotMqttQos) : BOOL  [EnsureSubscriptions]
//   Tc3_IotBase.TcIotMqttQos.AtLeastOnceDelivery   -> enum QoS 1                       [EnsureSubscriptions]
//   FB_IotMqttMessageQueue.nQueuedMessages : UDINT                                     [DrainOneMessage]
//   FB_IotMqttMessageQueue.Dequeue(fbMessage := FB_IotMqttMessage) : BOOL               [DrainOneMessage]
//   FB_IotMqttMessage.GetTopic(pTopic := PVOID, nTopicSize := UDINT) : BOOL            [DrainOneMessage]
//   FB_IotMqttMessage.GetPayload(pPayload := PVOID, nPayloadSize := UDINT,
//                                bSetNullTermination := BOOL) : BOOL                   [DrainOneMessage]
//
// Este FB e SOMENTE subscriber: NUNCA chama Publish. Nao ha teste unitario
// (precisa de um broker real) - validacao de runtime na bancada da Task 15.

bNewMessage := FALSE;

// -- desabilitado: derruba a conexao e zera o handshake de assinaturas --
IF NOT bEnable THEN
	fbMqtt.Execute(bConnect := FALSE);
	bConnected    := FALSE;
	bWasConnected := FALSE;
	bSubEstoque   := FALSE;
	bSubEventos   := FALSE;
	RETURN;
END_IF

// -- parametrizacao unica (host / porta / credenciais / TLS) --
IF NOT bParamsSet THEN
	ApplyBrokerParams();
	bParamsSet := TRUE;
END_IF

// -- conexao ciclica --
fbMqtt.Execute(bConnect := TRUE);
bConnected := fbMqtt.bConnected;

// -- contagem de reconexoes; a queda invalida as assinaturas --
IF bWasConnected AND NOT bConnected THEN
	nReconnectCount := nReconnectCount + 1;
	bSubEstoque := FALSE;
	bSubEventos := FALSE;
END_IF
bWasConnected := bConnected;

// -- garante as 2 assinaturas, uma vez por conexao --
IF bConnected THEN
	EnsureSubscriptions();
END_IF

// -- drena no maximo UMA mensagem por ciclo --
DrainOneMessage();

METHOD PROTECTED ApplyBrokerParams : BOOL
// ISOLADO DE PROPOSITO: todo membro de configuracao do FB_IotMqttClient
// (sHostName / nHostPort / sClientId / stMQTT.* / stTLS.*) vive aqui.
// Se um nome mudar na lib instalada, corrige-se somente este metodo.
// Chamado uma unica vez (guarda bParamsSet no corpo principal).
ApplyBrokerParams := TRUE;

fbMqtt.sHostName := stConfig.sMqttHost;
fbMqtt.nHostPort := stConfig.nMqttPort;
fbMqtt.sClientId := 'dataflow-cx9240-historian';

IF stConfig.sMqttUser <> '' THEN
	fbMqtt.sUserName   := stConfig.sMqttUser;
	fbMqtt.sUserPassword := stConfig.sMqttPass;
END_IF

IF stConfig.bUseTls THEN
	fbMqtt.stTLS.sCA := stConfig.sCaCertPath;
END_IF

// Sem isso, ipMessageQueue fica 0 para sempre e DrainOneMessage nunca dequeue
// nada - bConnected pode ficar TRUE mesmo assim (conexao e fila sao independentes).
fbMqtt.ipMessageQueue := fbMsgQueue;
END_METHOD

METHOD PROTECTED DrainOneMessage : BOOL
// ISOLADO DE PROPOSITO: todo acesso a fila de mensagens do TF6701 vive aqui
// (fbMsgQueue / nQueuedMessages / Dequeue / GetTopic / GetPayload).
// Retira NO MAXIMO uma mensagem por ciclo -> contrapressao previsivel para o
// pipeline a jusante. Em sucesso: sTopic e sPayload validos e bNewMessage = TRUE
// por exatamente 1 ciclo (o corpo principal zera bNewMessage no inicio do ciclo).
DrainOneMessage := FALSE;

IF fbMsgQueue.nQueuedMessages = 0 THEN
	RETURN;
END_IF

IF fbMsgQueue.Dequeue(fbMessage := fbMessage) THEN
	fbMessage.GetTopic(pTopic := ADR(sTopic), nTopicSize := SIZEOF(sTopic));
	fbMessage.GetPayload(pPayload            := ADR(sPayload),
	                     nPayloadSize        := SIZEOF(sPayload) - 1,
	                     bSetNullTermination := TRUE);
	bNewMessage     := TRUE;
	DrainOneMessage := TRUE;
END_IF
END_METHOD

METHOD PROTECTED EnsureSubscriptions : BOOL
// ISOLADO DE PROPOSITO: todas as chamadas Subscribe do TF6701 vivem aqui.
// Assina cada topico uma unica vez; bSubEstoque / bSubEventos sao zerados a
// cada reconexao no corpo principal. Retorna TRUE quando as 2 assinaturas
// ja foram aceitas pelo broker. So e chamado com bConnected = TRUE.
IF NOT bSubEstoque THEN
	bSubEstoque := fbMqtt.Subscribe(sTopic := stConfig.sTopicEstoque,
	                                eQoS  := Tc3_IotBase.TcIotMqttQos.AtLeastOnceDelivery);
END_IF

IF NOT bSubEventos THEN
	bSubEventos := fbMqtt.Subscribe(sTopic := stConfig.sTopicEventos,
	                                eQoS  := Tc3_IotBase.TcIotMqttQos.AtLeastOnceDelivery);
END_IF

EnsureSubscriptions := bSubEstoque AND bSubEventos;
END_METHOD

END_FUNCTION_BLOCK
